LIN {E6POS: X 1201.000, Y -192.200, Z 553.000, A 0.000, B 90.000, C 0.000, E1 0.000, E2 0.0, E3 0.0, E4 0.0, E5 0.0, E6 0.0} C_DIS
LIN {E6POS: X 1201.000, Y -191.200, Z 553.000, A 0.000, B 90.000, C 0.000, E1 0.000, E2 0.0, E3 0.0, E4 0.0, E5 0.0, E6 0.0} C_DIS
LIN {E6POS: X 1201.000, Y -190.200, Z 553.000, A 0.000, B 90.000, C 0.000, E1 0.000, E2 0.0, E3 0.0, E4 0.0, E5 0.0, E6 0.0} C_DIS
LIN {E6POS: X 1201.000, Y -189.200, Z 553.000, A 0.000, B 90.000, C 0.000, E1 0.000, E2 0.0, E3 0.0, E4 0.0, E5 0.0, E6 0.0} C_DIS
LIN {E6POS: X 1201.000, Y -188.200, Z 553.000, A 0.000, B 90.000, C 0.000, E1 0.000, E2 0.0, E3 0.0, E4 0.0, E5 0.0, E6 0.0} C_DIS
LIN {E6POS: X 1201.000, Y -187.200, Z 553.000, A 0.000, B 90.000, C 0.000, E1 0.000, E2 0.0, E3 0.0, E4 0.0, E5 0.0, E6 0.0} C_DIS
LIN {E6POS: X 1201.000, Y -187.200, Z 553.000, A 0.000, B 90.000, C 0.000, E1 0.000, E2 0.0, E3 0.0, E4 0.0, E5 0.0, E6 0.0} C_DIS
LIN {E6POS: X 1200.000, Y -187.200, Z 553.000, A 0.000, B 90.000, C 0.000, E1 0.000, E2 0.0, E3 0.0, E4 0.0, E5 0.0, E6 0.0} C_DIS
LIN {E6POS: X 1199.000, Y -187.200, Z 553.000, A 0.000, B 90.000, C 0.000, E1 0.000, E2 0.0, E3 0.0, E4 0.0, E5 0.0, E6 0.0} C_DIS
LIN {E6POS: X 1198.000, Y -187.200, Z 553.000, A 0.000, B 90.000, C 0.000, E1 0.000, E2 0.0, E3 0.0, E4 0.0, E5 0.0, E6 0.0} C_DIS
LIN {E6POS: X 1197.000, Y -187.200, Z 553.000, A 0.000, B 90.000, C 0.000, E1 0.000, E2 0.0, E3 0.0, E4 0.0, E5 0.0, E6 0.0} C_DIS
LIN {E6POS: X 1196.000, Y -187.200, Z 553.000, A 0.000, B 90.000, C 0.000, E1 0.000, E2 0.0, E3 0.0, E4 0.0, E5 0.0, E6 0.0} C_DIS
LIN {E6POS: X 1196.000, Y -187.200, Z 553.000, A 0.000, B 90.000, C 0.000, E1 0.000, E2 0.0, E3 0.0, E4 0.0, E5 0.0, E6 0.0} C_DIS
LIN {E6POS: X 1196.000, Y -188.200, Z 553.000, A 0.000, B 90.000, C 0.000, E1 0.000, E2 0.0, E3 0.0, E4 0.0, E5 0.0, E6 0.0} C_DIS
LIN {E6POS: X 1196.000, Y -189.200, Z 553.000, A 0.000, B 90.000, C 0.000, E1 0.000, E2 0.0, E3 0.0, E4 0.0, E5 0.0, E6 0.0} C_DIS
LIN {E6POS: X 1196.000, Y -190.200, Z 553.000, A 0.000, B 90.000, C 0.000, E1 0.000, E2 0.0, E3 0.0, E4 0.0, E5 0.0, E6 0.0} C_DIS
LIN {E6POS: X 1196.000, Y -191.200, Z 553.000, A 0.000, B 90.000, C 0.000, E1 0.000, E2 0.0, E3 0.0, E4 0.0, E5 0.0, E6 0.0} C_DIS
LIN {E6POS: X 1196.000, Y -192.200, Z 553.000, A 0.000, B 90.000, C 0.000, E1 0.000, E2 0.0, E3 0.0, E4 0.0, E5 0.0, E6 0.0} C_DIS
LIN {E6POS: X 1196.000, Y -193.200, Z 553.000, A 0.000, B 90.000, C 0.000, E1 0.000, E2 0.0, E3 0.0, E4 0.0, E5 0.0, E6 0.0} C_DIS
LIN {E6POS: X 1196.000, Y -194.200, Z 553.000, A 0.000, B 90.000, C 0.000, E1 0.000, E2 0.0, E3 0.0, E4 0.0, E5 0.0, E6 0.0} C_DIS
LIN {E6POS: X 1196.000, Y -195.200, Z 553.000, A 0.000, B 90.000, C 0.000, E1 0.000, E2 0.0, E3 0.0, E4 0.0, E5 0.0, E6 0.0} C_DIS
LIN {E6POS: X 1196.000, Y -196.200, Z 553.000, A 0.000, B 90.000, C 0.000, E1 0.000, E2 0.0, E3 0.0, E4 0.0, E5 0.0, E6 0.0} C_DIS
LIN {E6POS: X 1196.000, Y -197.200, Z 553.000, A 0.000, B 90.000, C 0.000, E1 0.000, E2 0.0, E3 0.0, E4 0.0, E5 0.0, E6 0.0} C_DIS
LIN {E6POS: X 1196.000, Y -198.200, Z 553.000, A 0.000, B 90.000, C 0.000, E1 0.000, E2 0.0, E3 0.0, E4 0.0, E5 0.0, E6 0.0} C_DIS
LIN {E6POS: X 1196.000, Y -199.200, Z 553.000, A 0.000, B 90.000, C 0.000, E1 0.000, E2 0.0, E3 0.0, E4 0.0, E5 0.0, E6 0.0} C_DIS
LIN {E6POS: X 1196.000, Y -200.200, Z 553.000, A 0.000, B 90.000, C 0.000, E1 0.000, E2 0.0, E3 0.0, E4 0.0, E5 0.0, E6 0.0} C_DIS
LIN {E6POS: X 1196.000, Y -201.200, Z 553.000, A 0.000, B 90.000, C 0.000, E1 0.000, E2 0.0, E3 0.0, E4 0.0, E5 0.0, E6 0.0} C_DIS
LIN {E6POS: X 1196.000, Y -202.200, Z 553.000, A 0.000, B 90.000, C 0.000, E1 0.000, E2 0.0, E3 0.0, E4 0.0, E5 0.0, E6 0.0} C_DIS
LIN {E6POS: X 1196.000, Y -203.200, Z 553.000, A 0.000, B 90.000, C 0.000, E1 0.000, E2 0.0, E3 0.0, E4 0.0, E5 0.0, E6 0.0} C_DIS
LIN {E6POS: X 1196.000, Y -204.200, Z 553.000, A 0.000, B 90.000, C 0.000, E1 0.000, E2 0.0, E3 0.0, E4 0.0, E5 0.0, E6 0.0} C_DIS
LIN {E6POS: X 1196.000, Y -205.200, Z 553.000, A 0.000, B 90.000, C 0.000, E1 0.000, E2 0.0, E3 0.0, E4 0.0, E5 0.0, E6 0.0} C_DIS
LIN {E6POS: X 1196.000, Y -206.200, Z 553.000, A 0.000, B 90.000, C 0.000, E1 0.000, E2 0.0, E3 0.0, E4 0.0, E5 0.0, E6 0.0} C_DIS
LIN {E6POS: X 1196.000, Y -207.200, Z 553.000, A 0.000, B 90.000, C 0.000, E1 0.000, E2 0.0, E3 0.0, E4 0.0, E5 0.0, E6 0.0} C_DIS
LIN {E6POS: X 1196.000, Y -208.200, Z 553.000, A 0.000, B 90.000, C 0.000, E1 0.000, E2 0.0, E3 0.0, E4 0.0, E5 0.0, E6 0.0} C_DIS
LIN {E6POS: X 1196.000, Y -209.200, Z 553.000, A 0.000, B 90.000, C 0.000, E1 0.000, E2 0.0, E3 0.0, E4 0.0, E5 0.0, E6 0.0} C_DIS
LIN {E6POS: X 1196.000, Y -210.200, Z 553.000, A 0.000, B 90.000, C 0.000, E1 0.000, E2 0.0, E3 0.0, E4 0.0, E5 0.0, E6 0.0} C_DIS
LIN {E6POS: X 1196.000, Y -211.200, Z 553.000, A 0.000, B 90.000, C 0.000, E1 0.000, E2 0.0, E3 0.0, E4 0.0, E5 0.0, E6 0.0} C_DIS
LIN {E6POS: X 1196.000, Y -212.200, Z 553.000, A 0.000, B 90.000, C 0.000, E1 0.000, E2 0.0, E3 0.0, E4 0.0, E5 0.0, E6 0.0} C_DIS
LIN {E6POS: X 1196.000, Y -213.200, Z 553.000, A 0.000, B 90.000, C 0.000, E1 0.000, E2 0.0, E3 0.0, E4 0.0, E5 0.0, E6 0.0} C_DIS
LIN {E6POS: X 1196.000, Y -214.200, Z 553.000, A 0.000, B 90.000, C 0.000, E1 0.000, E2 0.0, E3 0.0, E4 0.0, E5 0.0, E6 0.0} C_DIS
LIN {E6POS: X 1196.000, Y -215.200, Z 553.000, A 0.000, B 90.000, C 0.000, E1 0.000, E2 0.0, E3 0.0, E4 0.0, E5 0.0, E6 0.0} C_DIS
LIN {E6POS: X 1196.000, Y -216.200, Z 553.000, A 0.000, B 90.000, C 0.000, E1 0.000, E2 0.0, E3 0.0, E4 0.0, E5 0.0, E6 0.0} C_DIS
LIN {E6POS: X 1196.000, Y -217.200, Z 553.000, A 0.000, B 90.000, C 0.000, E1 0.000, E2 0.0, E3 0.0, E4 0.0, E5 0.0, E6 0.0} C_DIS
LIN {E6POS: X 1196.000, Y -218.200, Z 553.000, A 0.000, B 90.000, C 0.000, E1 0.000, E2 0.0, E3 0.0, E4 0.0, E5 0.0, E6 0.0} C_DIS
LIN {E6POS: X 1196.000, Y -219.200, Z 553.000, A 0.000, B 90.000, C 0.000, E1 0.000, E2 0.0, E3 0.0, E4 0.0, E5 0.0, E6 0.0} C_DIS
LIN {E6POS: X 1196.000, Y -220.200, Z 553.000, A 0.000, B 90.000, C 0.000, E1 0.000, E2 0.0, E3 0.0, E4 0.0, E5 0.0, E6 0.0} C_DIS
LIN {E6POS: X 1196.000, Y -221.200, Z 553.000, A 0.000, B 90.000, C 0.000, E1 0.000, E2 0.0, E3 0.0, E4 0.0, E5 0.0, E6 0.0} C_DIS
LIN {E6POS: X 1196.000, Y -222.200, Z 553.000, A 0.000, B 90.000, C 0.000, E1 0.000, E2 0.0, E3 0.0, E4 0.0, E5 0.0, E6 0.0} C_DIS
LIN {E6POS: X 1196.000, Y -223.200, Z 553.000, A 0.000, B 90.000, C 0.000, E1 0.000, E2 0.0, E3 0.0, E4 0.0, E5 0.0, E6 0.0} C_DIS
LIN {E6POS: X 1196.000, Y -224.200, Z 553.000, A 0.000, B 90.000, C 0.000, E1 0.000, E2 0.0, E3 0.0, E4 0.0, E5 0.0, E6 0.0} C_DIS
LIN {E6POS: X 1196.000, Y -225.200, Z 553.000, A 0.000, B 90.000, C 0.000, E1 0.000, E2 0.0, E3 0.0, E4 0.0, E5 0.0, E6 0.0} C_DIS
LIN {E6POS: X 1196.000, Y -226.200, Z 553.000, A 0.000, B 90.000, C 0.000, E1 0.000, E2 0.0, E3 0.0, E4 0.0, E5 0.0, E6 0.0} C_DIS
LIN {E6POS: X 1196.000, Y -227.200, Z 553.000, A 0.000, B 90.000, C 0.000, E1 0.000, E2 0.0, E3 0.0, E4 0.0, E5 0.0, E6 0.0} C_DIS
LIN {E6POS: X 1196.000, Y -228.200, Z 553.000, A 0.000, B 90.000, C 0.000, E1 0.000, E2 0.0, E3 0.0, E4 0.0, E5 0.0, E6 0.0} C_DIS
LIN {E6POS: X 1196.000, Y -229.200, Z 553.000, A 0.000, B 90.000, C 0.000, E1 0.000, E2 0.0, E3 0.0, E4 0.0, E5 0.0, E6 0.0} C_DIS
LIN {E6POS: X 1196.000, Y -230.200, Z 553.000, A 0.000, B 90.000, C 0.000, E1 0.000, E2 0.0, E3 0.0, E4 0.0, E5 0.0, E6 0.0} C_DIS
LIN {E6POS: X 1196.000, Y -231.200, Z 553.000, A 0.000, B 90.000, C 0.000, E1 0.000, E2 0.0, E3 0.0, E4 0.0, E5 0.0, E6 0.0} C_DIS
LIN {E6POS: X 1196.000, Y -232.200, Z 553.000, A 0.000, B 90.000, C 0.000, E1 0.000, E2 0.0, E3 0.0, E4 0.0, E5 0.0, E6 0.0} C_DIS
LIN {E6POS: X 1196.000, Y -233.200, Z 553.000, A 0.000, B 90.000, C 0.000, E1 0.000, E2 0.0, E3 0.0, E4 0.0, E5 0.0, E6 0.0} C_DIS
LIN {E6POS: X 1196.000, Y -234.200, Z 553.000, A 0.000, B 90.000, C 0.000, E1 0.000, E2 0.0, E3 0.0, E4 0.0, E5 0.0, E6 0.0} C_DIS
LIN {E6POS: X 1196.000, Y -235.200, Z 553.000, A 0.000, B 90.000, C 0.000, E1 0.000, E2 0.0, E3 0.0, E4 0.0, E5 0.0, E6 0.0} C_DIS
LIN {E6POS: X 1196.000, Y -236.200, Z 553.000, A 0.000, B 90.000, C 0.000, E1 0.000, E2 0.0, E3 0.0, E4 0.0, E5 0.0, E6 0.0} C_DIS
LIN {E6POS: X 1196.000, Y -237.200, Z 553.000, A 0.000, B 90.000, C 0.000, E1 0.000, E2 0.0, E3 0.0, E4 0.0, E5 0.0, E6 0.0} C_DIS
LIN {E6POS: X 1196.000, Y -237.200, Z 554.000, A 0.000, B 90.000, C 0.000, E1 0.000, E2 0.0, E3 0.0, E4 0.0, E5 0.0, E6 0.0} C_DIS
LIN {E6POS: X 1197.000, Y -237.200, Z 554.000, A 0.000, B 90.000, C 0.000, E1 0.000, E2 0.0, E3 0.0, E4 0.0, E5 0.0, E6 0.0} C_DIS
LIN {E6POS: X 1198.000, Y -237.200, Z 554.000, A 0.000, B 90.000, C 0.000, E1 0.000, E2 0.0, E3 0.0, E4 0.0, E5 0.0, E6 0.0} C_DIS
LIN {E6POS: X 1199.000, Y -237.200, Z 554.000, A 0.000, B 90.000, C 0.000, E1 0.000, E2 0.0, E3 0.0, E4 0.0, E5 0.0, E6 0.0} C_DIS
LIN {E6POS: X 1200.000, Y -237.200, Z 554.000, A 0.000, B 90.000, C 0.000, E1 0.000, E2 0.0, E3 0.0, E4 0.0, E5 0.0, E6 0.0} C_DIS
LIN {E6POS: X 1201.000, Y -237.200, Z 554.000, A 0.000, B 90.000, C 0.000, E1 0.000, E2 0.0, E3 0.0, E4 0.0, E5 0.0, E6 0.0} C_DIS
LIN {E6POS: X 1201.000, Y -237.200, Z 554.000, A 0.000, B 90.000, C 0.000, E1 0.000, E2 0.0, E3 0.0, E4 0.0, E5 0.0, E6 0.0} C_DIS
LIN {E6POS: X 1201.000, Y -236.200, Z 554.000, A 0.000, B 90.000, C 0.000, E1 0.000, E2 0.0, E3 0.0, E4 0.0, E5 0.0, E6 0.0} C_DIS
LIN {E6POS: X 1201.000, Y -235.200, Z 554.000, A 0.000, B 90.000, C 0.000, E1 0.000, E2 0.0, E3 0.0, E4 0.0, E5 0.0, E6 0.0} C_DIS
LIN {E6POS: X 1201.000, Y -234.200, Z 554.000, A 0.000, B 90.000, C 0.000, E1 0.000, E2 0.0, E3 0.0, E4 0.0, E5 0.0, E6 0.0} C_DIS
LIN {E6POS: X 1201.000, Y -233.200, Z 554.000, A 0.000, B 90.000, C 0.000, E1 0.000, E2 0.0, E3 0.0, E4 0.0, E5 0.0, E6 0.0} C_DIS
LIN {E6POS: X 1201.000, Y -232.200, Z 554.000, A 0.000, B 90.000, C 0.000, E1 0.000, E2 0.0, E3 0.0, E4 0.0, E5 0.0, E6 0.0} C_DIS
LIN {E6POS: X 1201.000, Y -231.200, Z 554.000, A 0.000, B 90.000, C 0.000, E1 0.000, E2 0.0, E3 0.0, E4 0.0, E5 0.0, E6 0.0} C_DIS
LIN {E6POS: X 1201.000, Y -230.200, Z 554.000, A 0.000, B 90.000, C 0.000, E1 0.000, E2 0.0, E3 0.0, E4 0.0, E5 0.0, E6 0.0} C_DIS
LIN {E6POS: X 1201.000, Y -229.200, Z 554.000, A 0.000, B 90.000, C 0.000, E1 0.000, E2 0.0, E3 0.0, E4 0.0, E5 0.0, E6 0.0} C_DIS
LIN {E6POS: X 1201.000, Y -228.200, Z 554.000, A 0.000, B 90.000, C 0.000, E1 0.000, E2 0.0, E3 0.0, E4 0.0, E5 0.0, E6 0.0} C_DIS
LIN {E6POS: X 1201.000, Y -227.200, Z 554.000, A 0.000, B 90.000, C 0.000, E1 0.000, E2 0.0, E3 0.0, E4 0.0, E5 0.0, E6 0.0} C_DIS
LIN {E6POS: X 1201.000, Y -226.200, Z 554.000, A 0.000, B 90.000, C 0.000, E1 0.000, E2 0.0, E3 0.0, E4 0.0, E5 0.0, E6 0.0} C_DIS
LIN {E6POS: X 1201.000, Y -225.200, Z 554.000, A 0.000, B 90.000, C 0.000, E1 0.000, E2 0.0, E3 0.0, E4 0.0, E5 0.0, E6 0.0} C_DIS
LIN {E6POS: X 1201.000, Y -224.200, Z 554.000, A 0.000, B 90.000, C 0.000, E1 0.000, E2 0.0, E3 0.0, E4 0.0, E5 0.0, E6 0.0} C_DIS
LIN {E6POS: X 1201.000, Y -223.200, Z 554.000, A 0.000, B 90.000, C 0.000, E1 0.000, E2 0.0, E3 0.0, E4 0.0, E5 0.0, E6 0.0} C_DIS
LIN {E6POS: X 1201.000, Y -222.200, Z 554.000, A 0.000, B 90.000, C 0.000, E1 0.000, E2 0.0, E3 0.0, E4 0.0, E5 0.0, E6 0.0} C_DIS
LIN {E6POS: X 1201.000, Y -221.200, Z 554.000, A 0.000, B 90.000, C 0.000, E1 0.000, E2 0.0, E3 0.0, E4 0.0, E5 0.0, E6 0.0} C_DIS
LIN {E6POS: X 1201.000, Y -220.200, Z 554.000, A 0.000, B 90.000, C 0.000, E1 0.000, E2 0.0, E3 0.0, E4 0.0, E5 0.0, E6 0.0} C_DIS
LIN {E6POS: X 1201.000, Y -219.200, Z 554.000, A 0.000, B 90.000, C 0.000, E1 0.000, E2 0.0, E3 0.0, E4 0.0, E5 0.0, E6 0.0} C_DIS
LIN {E6POS: X 1201.000, Y -218.200, Z 554.000, A 0.000, B 90.000, C 0.000, E1 0.000, E2 0.0, E3 0.0, E4 0.0, E5 0.0, E6 0.0} C_DIS
LIN {E6POS: X 1201.000, Y -217.200, Z 554.000, A 0.000, B 90.000, C 0.000, E1 0.000, E2 0.0, E3 0.0, E4 0.0, E5 0.0, E6 0.0} C_DIS
LIN {E6POS: X 1201.000, Y -216.200, Z 554.000, A 0.000, B 90.000, C 0.000, E1 0.000, E2 0.0, E3 0.0, E4 0.0, E5 0.0, E6 0.0} C_DIS
LIN {E6POS: X 1201.000, Y -215.200, Z 554.000, A 0.000, B 90.000, C 0.000, E1 0.000, E2 0.0, E3 0.0, E4 0.0, E5 0.0, E6 0.0} C_DIS
LIN {E6POS: X 1201.000, Y -214.200, Z 554.000, A 0.000, B 90.000, C 0.000, E1 0.000, E2 0.0, E3 0.0, E4 0.0, E5 0.0, E6 0.0} C_DIS
LIN {E6POS: X 1201.000, Y -213.200, Z 554.000, A 0.000, B 90.000, C 0.000, E1 0.000, E2 0.0, E3 0.0, E4 0.0, E5 0.0, E6 0.0} C_DIS
LIN {E6POS: X 1201.000, Y -212.200, Z 554.000, A 0.000, B 90.000, C 0.000, E1 0.000, E2 0.0, E3 0.0, E4 0.0, E5 0.0, E6 0.0} C_DIS
LIN {E6POS: X 1201.000, Y -211.200, Z 554.000, A 0.000, B 90.000, C 0.000, E1 0.000, E2 0.0, E3 0.0, E4 0.0, E5 0.0, E6 0.0} C_DIS
LIN {E6POS: X 1201.000, Y -210.200, Z 554.000, A 0.000, B 90.000, C 0.000, E1 0.000, E2 0.0, E3 0.0, E4 0.0, E5 0.0, E6 0.0} C_DIS
LIN {E6POS: X 1201.000, Y -209.200, Z 554.000, A 0.000, B 90.000, C 0.000, E1 0.000, E2 0.0, E3 0.0, E4 0.0, E5 0.0, E6 0.0} C_DIS
LIN {E6POS: X 1201.000, Y -208.200, Z 554.000, A 0.000, B 90.000, C 0.000, E1 0.000, E2 0.0, E3 0.0, E4 0.0, E5 0.0, E6 0.0} C_DIS
LIN {E6POS: X 1201.000, Y -207.200, Z 554.000, A 0.000, B 90.000, C 0.000, E1 0.000, E2 0.0, E3 0.0, E4 0.0, E5 0.0, E6 0.0} C_DIS
LIN {E6POS: X 1201.000, Y -206.200, Z 554.000, A 0.000, B 90.000, C 0.000, E1 0.000, E2 0.0, E3 0.0, E4 0.0, E5 0.0, E6 0.0} C_DIS
LIN {E6POS: X 1201.000, Y -205.200, Z 554.000, A 0.000, B 90.000, C 0.000, E1 0.000, E2 0.0, E3 0.0, E4 0.0, E5 0.0, E6 0.0} C_DIS
LIN {E6POS: X 1201.000, Y -204.200, Z 554.000, A 0.000, B 90.000, C 0.000, E1 0.000, E2 0.0, E3 0.0, E4 0.0, E5 0.0, E6 0.0} C_DIS
LIN {E6POS: X 1201.000, Y -203.200, Z 554.000, A 0.000, B 90.000, C 0.000, E1 0.000, E2 0.0, E3 0.0, E4 0.0, E5 0.0, E6 0.0} C_DIS
LIN {E6POS: X 1201.000, Y -202.200, Z 554.000, A 0.000, B 90.000, C 0.000, E1 0.000, E2 0.0, E3 0.0, E4 0.0, E5 0.0, E6 0.0} C_DIS
LIN {E6POS: X 1201.000, Y -201.200, Z 554.000, A 0.000, B 90.000, C 0.000, E1 0.000, E2 0.0, E3 0.0, E4 0.0, E5 0.0, E6 0.0} C_DIS
LIN {E6POS: X 1201.000, Y -200.200, Z 554.000, A 0.000, B 90.000, C 0.000, E1 0.000, E2 0.0, E3 0.0, E4 0.0, E5 0.0, E6 0.0} C_DIS
LIN {E6POS: X 1201.000, Y -199.200, Z 554.000, A 0.000, B 90.000, C 0.000, E1 0.000, E2 0.0, E3 0.0, E4 0.0, E5 0.0, E6 0.0} C_DIS
LIN {E6POS: X 1201.000, Y -198.200, Z 554.000, A 0.000, B 90.000, C 0.000, E1 0.000, E2 0.0, E3 0.0, E4 0.0, E5 0.0, E6 0.0} C_DIS
LIN {E6POS: X 1201.000, Y -197.200, Z 554.000, A 0.000, B 90.000, C 0.000, E1 0.000, E2 0.0, E3 0.0, E4 0.0, E5 0.0, E6 0.0} C_DIS
LIN {E6POS: X 1201.000, Y -196.200, Z 554.000, A 0.000, B 90.000, C 0.000, E1 0.000, E2 0.0, E3 0.0, E4 0.0, E5 0.0, E6 0.0} C_DIS
LIN {E6POS: X 1201.000, Y -195.200, Z 554.000, A 0.000, B 90.000, C 0.000, E1 0.000, E2 0.0, E3 0.0, E4 0.0, E5 0.0, E6 0.0} C_DIS
LIN {E6POS: X 1201.000, Y -194.200, Z 554.000, A 0.000, B 90.000, C 0.000, E1 0.000, E2 0.0, E3 0.0, E4 0.0, E5 0.0, E6 0.0} C_DIS
LIN {E6POS: X 1201.000, Y -193.200, Z 554.000, A 0.000, B 90.000, C 0.000, E1 0.000, E2 0.0, E3 0.0, E4 0.0, E5 0.0, E6 0.0} C_DIS
LIN {E6POS: X 1201.000, Y -192.200, Z 554.000, A 0.000, B 90.000, C 0.000, E1 0.000, E2 0.0, E3 0.0, E4 0.0, E5 0.0, E6 0.0} C_DIS
LIN {E6POS: X 1201.000, Y -191.200, Z 554.000, A 0.000, B 90.000, C 0.000, E1 0.000, E2 0.0, E3 0.0, E4 0.0, E5 0.0, E6 0.0} C_DIS
LIN {E6POS: X 1201.000, Y -190.200, Z 554.000, A 0.000, B 90.000, C 0.000, E1 0.000, E2 0.0, E3 0.0, E4 0.0, E5 0.0, E6 0.0} C_DIS
LIN {E6POS: X 1201.000, Y -189.200, Z 554.000, A 0.000, B 90.000, C 0.000, E1 0.000, E2 0.0, E3 0.0, E4 0.0, E5 0.0, E6 0.0} C_DIS
LIN {E6POS: X 1201.000, Y -188.200, Z 554.000, A 0.000, B 90.000, C 0.000, E1 0.000, E2 0.0, E3 0.0, E4 0.0, E5 0.0, E6 0.0} C_DIS
LIN {E6POS: X 1201.000, Y -187.200, Z 554.000, A 0.000, B 90.000, C 0.000, E1 0.000, E2 0.0, E3 0.0, E4 0.0, E5 0.0, E6 0.0} C_DIS
LIN {E6POS: X 1201.000, Y -187.200, Z 554.000, A 0.000, B 90.000, C 0.000, E1 0.000, E2 0.0, E3 0.0, E4 0.0, E5 0.0, E6 0.0} C_DIS
LIN {E6POS: X 1200.000, Y -187.200, Z 554.000, A 0.000, B 90.000, C 0.000, E1 0.000, E2 0.0, E3 0.0, E4 0.0, E5 0.0, E6 0.0} C_DIS
LIN {E6POS: X 1199.000, Y -187.200, Z 554.000, A 0.000, B 90.000, C 0.000, E1 0.000, E2 0.0, E3 0.0, E4 0.0, E5 0.0, E6 0.0} C_DIS
LIN {E6POS: X 1198.000, Y -187.200, Z 554.000, A 0.000, B 90.000, C 0.000, E1 0.000, E2 0.0, E3 0.0, E4 0.0, E5 0.0, E6 0.0} C_DIS
LIN {E6POS: X 1197.000, Y -187.200, Z 554.000, A 0.000, B 90.000, C 0.000, E1 0.000, E2 0.0, E3 0.0, E4 0.0, E5 0.0, E6 0.0} C_DIS
LIN {E6POS: X 1196.000, Y -187.200, Z 554.000, A 0.000, B 90.000, C 0.000, E1 0.000, E2 0.0, E3 0.0, E4 0.0, E5 0.0, E6 0.0} C_DIS
LIN {E6POS: X 1196.000, Y -187.200, Z 554.000, A 0.000, B 90.000, C 0.000, E1 0.000, E2 0.0, E3 0.0, E4 0.0, E5 0.0, E6 0.0} C_DIS
LIN {E6POS: X 1196.000, Y -188.200, Z 554.000, A 0.000, B 90.000, C 0.000, E1 0.000, E2 0.0, E3 0.0, E4 0.0, E5 0.0, E6 0.0} C_DIS
LIN {E6POS: X 1196.000, Y -189.200, Z 554.000, A 0.000, B 90.000, C 0.000, E1 0.000, E2 0.0, E3 0.0, E4 0.0, E5 0.0, E6 0.0} C_DIS
LIN {E6POS: X 1196.000, Y -190.200, Z 554.000, A 0.000, B 90.000, C 0.000, E1 0.000, E2 0.0, E3 0.0, E4 0.0, E5 0.0, E6 0.0} C_DIS
LIN {E6POS: X 1196.000, Y -191.200, Z 554.000, A 0.000, B 90.000, C 0.000, E1 0.000, E2 0.0, E3 0.0, E4 0.0, E5 0.0, E6 0.0} C_DIS
LIN {E6POS: X 1196.000, Y -192.200, Z 554.000, A 0.000, B 90.000, C 0.000, E1 0.000, E2 0.0, E3 0.0, E4 0.0, E5 0.0, E6 0.0} C_DIS
LIN {E6POS: X 1196.000, Y -193.200, Z 554.000, A 0.000, B 90.000, C 0.000, E1 0.000, E2 0.0, E3 0.0, E4 0.0, E5 0.0, E6 0.0} C_DIS
LIN {E6POS: X 1196.000, Y -194.200, Z 554.000, A 0.000, B 90.000, C 0.000, E1 0.000, E2 0.0, E3 0.0, E4 0.0, E5 0.0, E6 0.0} C_DIS
LIN {E6POS: X 1196.000, Y -195.200, Z 554.000, A 0.000, B 90.000, C 0.000, E1 0.000, E2 0.0, E3 0.0, E4 0.0, E5 0.0, E6 0.0} C_DIS
LIN {E6POS: X 1196.000, Y -196.200, Z 554.000, A 0.000, B 90.000, C 0.000, E1 0.000, E2 0.0, E3 0.0, E4 0.0, E5 0.0, E6 0.0} C_DIS
LIN {E6POS: X 1196.000, Y -197.200, Z 554.000, A 0.000, B 90.000, C 0.000, E1 0.000, E2 0.0, E3 0.0, E4 0.0, E5 0.0, E6 0.0} C_DIS
LIN {E6POS: X 1196.000, Y -198.200, Z 554.000, A 0.000, B 90.000, C 0.000, E1 0.000, E2 0.0, E3 0.0, E4 0.0, E5 0.0, E6 0.0} C_DIS
LIN {E6POS: X 1196.000, Y -199.200, Z 554.000, A 0.000, B 90.000, C 0.000, E1 0.000, E2 0.0, E3 0.0, E4 0.0, E5 0.0, E6 0.0} C_DIS
LIN {E6POS: X 1196.000, Y -200.200, Z 554.000, A 0.000, B 90.000, C 0.000, E1 0.000, E2 0.0, E3 0.0, E4 0.0, E5 0.0, E6 0.0} C_DIS
LIN {E6POS: X 1196.000, Y -201.200, Z 554.000, A 0.000, B 90.000, C 0.000, E1 0.000, E2 0.0, E3 0.0, E4 0.0, E5 0.0, E6 0.0} C_DIS
LIN {E6POS: X 1196.000, Y -202.200, Z 554.000, A 0.000, B 90.000, C 0.000, E1 0.000, E2 0.0, E3 0.0, E4 0.0, E5 0.0, E6 0.0} C_DIS
LIN {E6POS: X 1196.000, Y -203.200, Z 554.000, A 0.000, B 90.000, C 0.000, E1 0.000, E2 0.0, E3 0.0, E4 0.0, E5 0.0, E6 0.0} C_DIS
LIN {E6POS: X 1196.000, Y -204.200, Z 554.000, A 0.000, B 90.000, C 0.000, E1 0.000, E2 0.0, E3 0.0, E4 0.0, E5 0.0, E6 0.0} C_DIS
LIN {E6POS: X 1196.000, Y -205.200, Z 554.000, A 0.000, B 90.000, C 0.000, E1 0.000, E2 0.0, E3 0.0, E4 0.0, E5 0.0, E6 0.0} C_DIS
LIN {E6POS: X 1196.000, Y -206.200, Z 554.000, A 0.000, B 90.000, C 0.000, E1 0.000, E2 0.0, E3 0.0, E4 0.0, E5 0.0, E6 0.0} C_DIS
LIN {E6POS: X 1196.000, Y -207.200, Z 554.000, A 0.000, B 90.000, C 0.000, E1 0.000, E2 0.0, E3 0.0, E4 0.0, E5 0.0, E6 0.0} C_DIS
LIN {E6POS: X 1196.000, Y -208.200, Z 554.000, A 0.000, B 90.000, C 0.000, E1 0.000, E2 0.0, E3 0.0, E4 0.0, E5 0.0, E6 0.0} C_DIS
LIN {E6POS: X 1196.000, Y -209.200, Z 554.000, A 0.000, B 90.000, C 0.000, E1 0.000, E2 0.0, E3 0.0, E4 0.0, E5 0.0, E6 0.0} C_DIS
LIN {E6POS: X 1196.000, Y -210.200, Z 554.000, A 0.000, B 90.000, C 0.000, E1 0.000, E2 0.0, E3 0.0, E4 0.0, E5 0.0, E6 0.0} C_DIS
LIN {E6POS: X 1196.000, Y -211.200, Z 554.000, A 0.000, B 90.000, C 0.000, E1 0.000, E2 0.0, E3 0.0, E4 0.0, E5 0.0, E6 0.0} C_DIS
LIN {E6POS: X 1196.000, Y -212.200, Z 554.000, A 0.000, B 90.000, C 0.000, E1 0.000, E2 0.0, E3 0.0, E4 0.0, E5 0.0, E6 0.0} C_DIS
LIN {E6POS: X 1196.000, Y -213.200, Z 554.000, A 0.000, B 90.000, C 0.000, E1 0.000, E2 0.0, E3 0.0, E4 0.0, E5 0.0, E6 0.0} C_DIS
LIN {E6POS: X 1196.000, Y -214.200, Z 554.000, A 0.000, B 90.000, C 0.000, E1 0.000, E2 0.0, E3 0.0, E4 0.0, E5 0.0, E6 0.0} C_DIS
LIN {E6POS: X 1196.000, Y -215.200, Z 554.000, A 0.000, B 90.000, C 0.000, E1 0.000, E2 0.0, E3 0.0, E4 0.0, E5 0.0, E6 0.0} C_DIS
LIN {E6POS: X 1196.000, Y -216.200, Z 554.000, A 0.000, B 90.000, C 0.000, E1 0.000, E2 0.0, E3 0.0, E4 0.0, E5 0.0, E6 0.0} C_DIS
LIN {E6POS: X 1196.000, Y -217.200, Z 554.000, A 0.000, B 90.000, C 0.000, E1 0.000, E2 0.0, E3 0.0, E4 0.0, E5 0.0, E6 0.0} C_DIS
LIN {E6POS: X 1196.000, Y -218.200, Z 554.000, A 0.000, B 90.000, C 0.000, E1 0.000, E2 0.0, E3 0.0, E4 0.0, E5 0.0, E6 0.0} C_DIS
LIN {E6POS: X 1196.000, Y -219.200, Z 554.000, A 0.000, B 90.000, C 0.000, E1 0.000, E2 0.0, E3 0.0, E4 0.0, E5 0.0, E6 0.0} C_DIS
LIN {E6POS: X 1196.000, Y -220.200, Z 554.000, A 0.000, B 90.000, C 0.000, E1 0.000, E2 0.0, E3 0.0, E4 0.0, E5 0.0, E6 0.0} C_DIS
LIN {E6POS: X 1196.000, Y -221.200, Z 554.000, A 0.000, B 90.000, C 0.000, E1 0.000, E2 0.0, E3 0.0, E4 0.0, E5 0.0, E6 0.0} C_DIS
LIN {E6POS: X 1196.000, Y -222.200, Z 554.000, A 0.000, B 90.000, C 0.000, E1 0.000, E2 0.0, E3 0.0, E4 0.0, E5 0.0, E6 0.0} C_DIS
LIN {E6POS: X 1196.000, Y -223.200, Z 554.000, A 0.000, B 90.000, C 0.000, E1 0.000, E2 0.0, E3 0.0, E4 0.0, E5 0.0, E6 0.0} C_DIS
LIN {E6POS: X 1196.000, Y -224.200, Z 554.000, A 0.000, B 90.000, C 0.000, E1 0.000, E2 0.0, E3 0.0, E4 0.0, E5 0.0, E6 0.0} C_DIS
LIN {E6POS: X 1196.000, Y -225.200, Z 554.000, A 0.000, B 90.000, C 0.000, E1 0.000, E2 0.0, E3 0.0, E4 0.0, E5 0.0, E6 0.0} C_DIS
LIN {E6POS: X 1196.000, Y -226.200, Z 554.000, A 0.000, B 90.000, C 0.000, E1 0.000, E2 0.0, E3 0.0, E4 0.0, E5 0.0, E6 0.0} C_DIS
LIN {E6POS: X 1196.000, Y -227.200, Z 554.000, A 0.000, B 90.000, C 0.000, E1 0.000, E2 0.0, E3 0.0, E4 0.0, E5 0.0, E6 0.0} C_DIS
LIN {E6POS: X 1196.000, Y -228.200, Z 554.000, A 0.000, B 90.000, C 0.000, E1 0.000, E2 0.0, E3 0.0, E4 0.0, E5 0.0, E6 0.0} C_DIS
LIN {E6POS: X 1196.000, Y -229.200, Z 554.000, A 0.000, B 90.000, C 0.000, E1 0.000, E2 0.0, E3 0.0, E4 0.0, E5 0.0, E6 0.0} C_DIS
LIN {E6POS: X 1196.000, Y -230.200, Z 554.000, A 0.000, B 90.000, C 0.000, E1 0.000, E2 0.0, E3 0.0, E4 0.0, E5 0.0, E6 0.0} C_DIS
LIN {E6POS: X 1196.000, Y -231.200, Z 554.000, A 0.000, B 90.000, C 0.000, E1 0.000, E2 0.0, E3 0.0, E4 0.0, E5 0.0, E6 0.0} C_DIS
LIN {E6POS: X 1196.000, Y -232.200, Z 554.000, A 0.000, B 90.000, C 0.000, E1 0.000, E2 0.0, E3 0.0, E4 0.0, E5 0.0, E6 0.0} C_DIS
LIN {E6POS: X 1196.000, Y -233.200, Z 554.000, A 0.000, B 90.000, C 0.000, E1 0.000, E2 0.0, E3 0.0, E4 0.0, E5 0.0, E6 0.0} C_DIS
LIN {E6POS: X 1196.000, Y -234.200, Z 554.000, A 0.000, B 90.000, C 0.000, E1 0.000, E2 0.0, E3 0.0, E4 0.0, E5 0.0, E6 0.0} C_DIS
LIN {E6POS: X 1196.000, Y -235.200, Z 554.000, A 0.000, B 90.000, C 0.000, E1 0.000, E2 0.0, E3 0.0, E4 0.0, E5 0.0, E6 0.0} C_DIS
LIN {E6POS: X 1196.000, Y -236.200, Z 554.000, A 0.000, B 90.000, C 0.000, E1 0.000, E2 0.0, E3 0.0, E4 0.0, E5 0.0, E6 0.0} C_DIS
LIN {E6POS: X 1196.000, Y -237.200, Z 554.000, A 0.000, B 90.000, C 0.000, E1 0.000, E2 0.0, E3 0.0, E4 0.0, E5 0.0, E6 0.0} C_DIS
LIN {E6POS: X 1196.000, Y -237.200, Z 555.000, A 0.000, B 90.000, C 0.000, E1 0.000, E2 0.0, E3 0.0, E4 0.0, E5 0.0, E6 0.0} C_DIS
LIN {E6POS: X 1197.000, Y -237.200, Z 555.000, A 0.000, B 90.000, C 0.000, E1 0.000, E2 0.0, E3 0.0, E4 0.0, E5 0.0, E6 0.0} C_DIS
LIN {E6POS: X 1198.000, Y -237.200, Z 555.000, A 0.000, B 90.000, C 0.000, E1 0.000, E2 0.0, E3 0.0, E4 0.0, E5 0.0, E6 0.0} C_DIS
LIN {E6POS: X 1199.000, Y -237.200, Z 555.000, A 0.000, B 90.000, C 0.000, E1 0.000, E2 0.0, E3 0.0, E4 0.0, E5 0.0, E6 0.0} C_DIS
LIN {E6POS: X 1200.000, Y -237.200, Z 555.000, A 0.000, B 90.000, C 0.000, E1 0.000, E2 0.0, E3 0.0, E4 0.0, E5 0.0, E6 0.0} C_DIS
LIN {E6POS: X 1201.000, Y -237.200, Z 555.000, A 0.000, B 90.000, C 0.000, E1 0.000, E2 0.0, E3 0.0, E4 0.0, E5 0.0, E6 0.0} C_DIS
LIN {E6POS: X 1201.000, Y -237.200, Z 555.000, A 0.000, B 90.000, C 0.000, E1 0.000, E2 0.0, E3 0.0, E4 0.0, E5 0.0, E6 0.0} C_DIS
LIN {E6POS: X 1201.000, Y -236.200, Z 555.000, A 0.000, B 90.000, C 0.000, E1 0.000, E2 0.0, E3 0.0, E4 0.0, E5 0.0, E6 0.0} C_DIS
LIN {E6POS: X 1201.000, Y -235.200, Z 555.000, A 0.000, B 90.000, C 0.000, E1 0.000, E2 0.0, E3 0.0, E4 0.0, E5 0.0, E6 0.0} C_DIS
LIN {E6POS: X 1201.000, Y -234.200, Z 555.000, A 0.000, B 90.000, C 0.000, E1 0.000, E2 0.0, E3 0.0, E4 0.0, E5 0.0, E6 0.0} C_DIS
LIN {E6POS: X 1201.000, Y -233.200, Z 555.000, A 0.000, B 90.000, C 0.000, E1 0.000, E2 0.0, E3 0.0, E4 0.0, E5 0.0, E6 0.0} C_DIS
LIN {E6POS: X 1201.000, Y -232.200, Z 555.000, A 0.000, B 90.000, C 0.000, E1 0.000, E2 0.0, E3 0.0, E4 0.0, E5 0.0, E6 0.0} C_DIS
LIN {E6POS: X 1201.000, Y -231.200, Z 555.000, A 0.000, B 90.000, C 0.000, E1 0.000, E2 0.0, E3 0.0, E4 0.0, E5 0.0, E6 0.0} C_DIS
LIN {E6POS: X 1201.000, Y -230.200, Z 555.000, A 0.000, B 90.000, C 0.000, E1 0.000, E2 0.0, E3 0.0, E4 0.0, E5 0.0, E6 0.0} C_DIS
LIN {E6POS: X 1201.000, Y -229.200, Z 555.000, A 0.000, B 90.000, C 0.000, E1 0.000, E2 0.0, E3 0.0, E4 0.0, E5 0.0, E6 0.0} C_DIS
LIN {E6POS: X 1201.000, Y -228.200, Z 555.000, A 0.000, B 90.000, C 0.000, E1 0.000, E2 0.0, E3 0.0, E4 0.0, E5 0.0, E6 0.0} C_DIS
LIN {E6POS: X 1201.000, Y -227.200, Z 555.000, A 0.000, B 90.000, C 0.000, E1 0.000, E2 0.0, E3 0.0, E4 0.0, E5 0.0, E6 0.0} C_DIS
LIN {E6POS: X 1201.000, Y -226.200, Z 555.000, A 0.000, B 90.000, C 0.000, E1 0.000, E2 0.0, E3 0.0, E4 0.0, E5 0.0, E6 0.0} C_DIS
LIN {E6POS: X 1201.000, Y -225.200, Z 555.000, A 0.000, B 90.000, C 0.000, E1 0.000, E2 0.0, E3 0.0, E4 0.0, E5 0.0, E6 0.0} C_DIS
LIN {E6POS: X 1201.000, Y -224.200, Z 555.000, A 0.000, B 90.000, C 0.000, E1 0.000, E2 0.0, E3 0.0, E4 0.0, E5 0.0, E6 0.0} C_DIS
LIN {E6POS: X 1201.000, Y -223.200, Z 555.000, A 0.000, B 90.000, C 0.000, E1 0.000, E2 0.0, E3 0.0, E4 0.0, E5 0.0, E6 0.0} C_DIS
LIN {E6POS: X 1201.000, Y -222.200, Z 555.000, A 0.000, B 90.000, C 0.000, E1 0.000, E2 0.0, E3 0.0, E4 0.0, E5 0.0, E6 0.0} C_DIS
LIN {E6POS: X 1201.000, Y -221.200, Z 555.000, A 0.000, B 90.000, C 0.000, E1 0.000, E2 0.0, E3 0.0, E4 0.0, E5 0.0, E6 0.0} C_DIS
LIN {E6POS: X 1201.000, Y -220.200, Z 555.000, A 0.000, B 90.000, C 0.000, E1 0.000, E2 0.0, E3 0.0, E4 0.0, E5 0.0, E6 0.0} C_DIS
LIN {E6POS: X 1201.000, Y -219.200, Z 555.000, A 0.000, B 90.000, C 0.000, E1 0.000, E2 0.0, E3 0.0, E4 0.0, E5 0.0, E6 0.0} C_DIS
LIN {E6POS: X 1201.000, Y -218.200, Z 555.000, A 0.000, B 90.000, C 0.000, E1 0.000, E2 0.0, E3 0.0, E4 0.0, E5 0.0, E6 0.0} C_DIS
LIN {E6POS: X 1201.000, Y -217.200, Z 555.000, A 0.000, B 90.000, C 0.000, E1 0.000, E2 0.0, E3 0.0, E4 0.0, E5 0.0, E6 0.0} C_DIS
LIN {E6POS: X 1201.000, Y -216.200, Z 555.000, A 0.000, B 90.000, C 0.000, E1 0.000, E2 0.0, E3 0.0, E4 0.0, E5 0.0, E6 0.0} C_DIS
LIN {E6POS: X 1201.000, Y -215.200, Z 555.000, A 0.000, B 90.000, C 0.000, E1 0.000, E2 0.0, E3 0.0, E4 0.0, E5 0.0, E6 0.0} C_DIS
LIN {E6POS: X 1201.000, Y -214.200, Z 555.000, A 0.000, B 90.000, C 0.000, E1 0.000, E2 0.0, E3 0.0, E4 0.0, E5 0.0, E6 0.0} C_DIS
LIN {E6POS: X 1201.000, Y -213.200, Z 555.000, A 0.000, B 90.000, C 0.000, E1 0.000, E2 0.0, E3 0.0, E4 0.0, E5 0.0, E6 0.0} C_DIS
LIN {E6POS: X 1201.000, Y -212.200, Z 555.000, A 0.000, B 90.000, C 0.000, E1 0.000, E2 0.0, E3 0.0, E4 0.0, E5 0.0, E6 0.0} C_DIS
LIN {E6POS: X 1201.000, Y -211.200, Z 555.000, A 0.000, B 90.000, C 0.000, E1 0.000, E2 0.0, E3 0.0, E4 0.0, E5 0.0, E6 0.0} C_DIS
LIN {E6POS: X 1201.000, Y -210.200, Z 555.000, A 0.000, B 90.000, C 0.000, E1 0.000, E2 0.0, E3 0.0, E4 0.0, E5 0.0, E6 0.0} C_DIS
LIN {E6POS: X 1201.000, Y -209.200, Z 555.000, A 0.000, B 90.000, C 0.000, E1 0.000, E2 0.0, E3 0.0, E4 0.0, E5 0.0, E6 0.0} C_DIS
LIN {E6POS: X 1201.000, Y -208.200, Z 555.000, A 0.000, B 90.000, C 0.000, E1 0.000, E2 0.0, E3 0.0, E4 0.0, E5 0.0, E6 0.0} C_DIS
LIN {E6POS: X 1201.000, Y -207.200, Z 555.000, A 0.000, B 90.000, C 0.000, E1 0.000, E2 0.0, E3 0.0, E4 0.0, E5 0.0, E6 0.0} C_DIS
LIN {E6POS: X 1201.000, Y -206.200, Z 555.000, A 0.000, B 90.000, C 0.000, E1 0.000, E2 0.0, E3 0.0, E4 0.0, E5 0.0, E6 0.0} C_DIS
LIN {E6POS: X 1201.000, Y -205.200, Z 555.000, A 0.000, B 90.000, C 0.000, E1 0.000, E2 0.0, E3 0.0, E4 0.0, E5 0.0, E6 0.0} C_DIS
LIN {E6POS: X 1201.000, Y -204.200, Z 555.000, A 0.000, B 90.000, C 0.000, E1 0.000, E2 0.0, E3 0.0, E4 0.0, E5 0.0, E6 0.0} C_DIS
LIN {E6POS: X 1201.000, Y -203.200, Z 555.000, A 0.000, B 90.000, C 0.000, E1 0.000, E2 0.0, E3 0.0, E4 0.0, E5 0.0, E6 0.0} C_DIS
LIN {E6POS: X 1201.000, Y -202.200, Z 555.000, A 0.000, B 90.000, C 0.000, E1 0.000, E2 0.0, E3 0.0, E4 0.0, E5 0.0, E6 0.0} C_DIS
LIN {E6POS: X 1201.000, Y -201.200, Z 555.000, A 0.000, B 90.000, C 0.000, E1 0.000, E2 0.0, E3 0.0, E4 0.0, E5 0.0, E6 0.0} C_DIS
LIN {E6POS: X 1201.000, Y -200.200, Z 555.000, A 0.000, B 90.000, C 0.000, E1 0.000, E2 0.0, E3 0.0, E4 0.0, E5 0.0, E6 0.0} C_DIS
LIN {E6POS: X 1201.000, Y -199.200, Z 555.000, A 0.000, B 90.000, C 0.000, E1 0.000, E2 0.0, E3 0.0, E4 0.0, E5 0.0, E6 0.0} C_DIS
LIN {E6POS: X 1201.000, Y -198.200, Z 555.000, A 0.000, B 90.000, C 0.000, E1 0.000, E2 0.0, E3 0.0, E4 0.0, E5 0.0, E6 0.0} C_DIS
LIN {E6POS: X 1201.000, Y -197.200, Z 555.000, A 0.000, B 90.000, C 0.000, E1 0.000, E2 0.0, E3 0.0, E4 0.0, E5 0.0, E6 0.0} C_DIS
LIN {E6POS: X 1201.000, Y -196.200, Z 555.000, A 0.000, B 90.000, C 0.000, E1 0.000, E2 0.0, E3 0.0, E4 0.0, E5 0.0, E6 0.0} C_DIS
LIN {E6POS: X 1201.000, Y -195.200, Z 555.000, A 0.000, B 90.000, C 0.000, E1 0.000, E2 0.0, E3 0.0, E4 0.0, E5 0.0, E6 0.0} C_DIS
LIN {E6POS: X 1201.000, Y -194.200, Z 555.000, A 0.000, B 90.000, C 0.000, E1 0.000, E2 0.0, E3 0.0, E4 0.0, E5 0.0, E6 0.0} C_DIS
LIN {E6POS: X 1201.000, Y -193.200, Z 555.000, A 0.000, B 90.000, C 0.000, E1 0.000, E2 0.0, E3 0.0, E4 0.0, E5 0.0, E6 0.0} C_DIS
LIN {E6POS: X 1201.000, Y -192.200, Z 555.000, A 0.000, B 90.000, C 0.000, E1 0.000, E2 0.0, E3 0.0, E4 0.0, E5 0.0, E6 0.0} C_DIS
LIN {E6POS: X 1201.000, Y -191.200, Z 555.000, A 0.000, B 90.000, C 0.000, E1 0.000, E2 0.0, E3 0.0, E4 0.0, E5 0.0, E6 0.0} C_DIS
LIN {E6POS: X 1201.000, Y -190.200, Z 555.000, A 0.000, B 90.000, C 0.000, E1 0.000, E2 0.0, E3 0.0, E4 0.0, E5 0.0, E6 0.0} C_DIS
LIN {E6POS: X 1201.000, Y -189.200, Z 555.000, A 0.000, B 90.000, C 0.000, E1 0.000, E2 0.0, E3 0.0, E4 0.0, E5 0.0, E6 0.0} C_DIS
LIN {E6POS: X 1201.000, Y -188.200, Z 555.000, A 0.000, B 90.000, C 0.000, E1 0.000, E2 0.0, E3 0.0, E4 0.0, E5 0.0, E6 0.0} C_DIS
LIN {E6POS: X 1201.000, Y -187.200, Z 555.000, A 0.000, B 90.000, C 0.000, E1 0.000, E2 0.0, E3 0.0, E4 0.0, E5 0.0, E6 0.0} C_DIS
LIN {E6POS: X 1201.000, Y -187.200, Z 555.000, A 0.000, B 90.000, C 0.000, E1 0.000, E2 0.0, E3 0.0, E4 0.0, E5 0.0, E6 0.0} C_DIS
LIN {E6POS: X 1200.000, Y -187.200, Z 555.000, A 0.000, B 90.000, C 0.000, E1 0.000, E2 0.0, E3 0.0, E4 0.0, E5 0.0, E6 0.0} C_DIS
LIN {E6POS: X 1199.000, Y -187.200, Z 555.000, A 0.000, B 90.000, C 0.000, E1 0.000, E2 0.0, E3 0.0, E4 0.0, E5 0.0, E6 0.0} C_DIS
LIN {E6POS: X 1198.000, Y -187.200, Z 555.000, A 0.000, B 90.000, C 0.000, E1 0.000, E2 0.0, E3 0.0, E4 0.0, E5 0.0, E6 0.0} C_DIS
LIN {E6POS: X 1197.000, Y -187.200, Z 555.000, A 0.000, B 90.000, C 0.000, E1 0.000, E2 0.0, E3 0.0, E4 0.0, E5 0.0, E6 0.0} C_DIS
LIN {E6POS: X 1196.000, Y -187.200, Z 555.000, A 0.000, B 90.000, C 0.000, E1 0.000, E2 0.0, E3 0.0, E4 0.0, E5 0.0, E6 0.0} C_DIS
LIN {E6POS: X 1196.000, Y -187.200, Z 555.000, A 0.000, B 90.000, C 0.000, E1 0.000, E2 0.0, E3 0.0, E4 0.0, E5 0.0, E6 0.0} C_DIS
LIN {E6POS: X 1196.000, Y -188.200, Z 555.000, A 0.000, B 90.000, C 0.000, E1 0.000, E2 0.0, E3 0.0, E4 0.0, E5 0.0, E6 0.0} C_DIS
LIN {E6POS: X 1196.000, Y -189.200, Z 555.000, A 0.000, B 90.000, C 0.000, E1 0.000, E2 0.0, E3 0.0, E4 0.0, E5 0.0, E6 0.0} C_DIS
LIN {E6POS: X 1196.000, Y -190.200, Z 555.000, A 0.000, B 90.000, C 0.000, E1 0.000, E2 0.0, E3 0.0, E4 0.0, E5 0.0, E6 0.0} C_DIS
LIN {E6POS: X 1196.000, Y -191.200, Z 555.000, A 0.000, B 90.000, C 0.000, E1 0.000, E2 0.0, E3 0.0, E4 0.0, E5 0.0, E6 0.0} C_DIS
LIN {E6POS: X 1196.000, Y -192.200, Z 555.000, A 0.000, B 90.000, C 0.000, E1 0.000, E2 0.0, E3 0.0, E4 0.0, E5 0.0, E6 0.0} C_DIS
LIN {E6POS: X 1196.000, Y -193.200, Z 555.000, A 0.000, B 90.000, C 0.000, E1 0.000, E2 0.0, E3 0.0, E4 0.0, E5 0.0, E6 0.0} C_DIS
LIN {E6POS: X 1196.000, Y -194.200, Z 555.000, A 0.000, B 90.000, C 0.000, E1 0.000, E2 0.0, E3 0.0, E4 0.0, E5 0.0, E6 0.0} C_DIS
LIN {E6POS: X 1196.000, Y -195.200, Z 555.000, A 0.000, B 90.000, C 0.000, E1 0.000, E2 0.0, E3 0.0, E4 0.0, E5 0.0, E6 0.0} C_DIS
LIN {E6POS: X 1196.000, Y -196.200, Z 555.000, A 0.000, B 90.000, C 0.000, E1 0.000, E2 0.0, E3 0.0, E4 0.0, E5 0.0, E6 0.0} C_DIS
LIN {E6POS: X 1196.000, Y -197.200, Z 555.000, A 0.000, B 90.000, C 0.000, E1 0.000, E2 0.0, E3 0.0, E4 0.0, E5 0.0, E6 0.0} C_DIS
LIN {E6POS: X 1196.000, Y -198.200, Z 555.000, A 0.000, B 90.000, C 0.000, E1 0.000, E2 0.0, E3 0.0, E4 0.0, E5 0.0, E6 0.0} C_DIS
LIN {E6POS: X 1196.000, Y -199.200, Z 555.000, A 0.000, B 90.000, C 0.000, E1 0.000, E2 0.0, E3 0.0, E4 0.0, E5 0.0, E6 0.0} C_DIS
LIN {E6POS: X 1196.000, Y -200.200, Z 555.000, A 0.000, B 90.000, C 0.000, E1 0.000, E2 0.0, E3 0.0, E4 0.0, E5 0.0, E6 0.0} C_DIS
LIN {E6POS: X 1196.000, Y -201.200, Z 555.000, A 0.000, B 90.000, C 0.000, E1 0.000, E2 0.0, E3 0.0, E4 0.0, E5 0.0, E6 0.0} C_DIS
LIN {E6POS: X 1196.000, Y -202.200, Z 555.000, A 0.000, B 90.000, C 0.000, E1 0.000, E2 0.0, E3 0.0, E4 0.0, E5 0.0, E6 0.0} C_DIS
LIN {E6POS: X 1196.000, Y -203.200, Z 555.000, A 0.000, B 90.000, C 0.000, E1 0.000, E2 0.0, E3 0.0, E4 0.0, E5 0.0, E6 0.0} C_DIS
LIN {E6POS: X 1196.000, Y -204.200, Z 555.000, A 0.000, B 90.000, C 0.000, E1 0.000, E2 0.0, E3 0.0, E4 0.0, E5 0.0, E6 0.0} C_DIS
LIN {E6POS: X 1196.000, Y -205.200, Z 555.000, A 0.000, B 90.000, C 0.000, E1 0.000, E2 0.0, E3 0.0, E4 0.0, E5 0.0, E6 0.0} C_DIS
LIN {E6POS: X 1196.000, Y -206.200, Z 555.000, A 0.000, B 90.000, C 0.000, E1 0.000, E2 0.0, E3 0.0, E4 0.0, E5 0.0, E6 0.0} C_DIS
LIN {E6POS: X 1196.000, Y -207.200, Z 555.000, A 0.000, B 90.000, C 0.000, E1 0.000, E2 0.0, E3 0.0, E4 0.0, E5 0.0, E6 0.0} C_DIS
LIN {E6POS: X 1196.000, Y -208.200, Z 555.000, A 0.000, B 90.000, C 0.000, E1 0.000, E2 0.0, E3 0.0, E4 0.0, E5 0.0, E6 0.0} C_DIS
LIN {E6POS: X 1196.000, Y -209.200, Z 555.000, A 0.000, B 90.000, C 0.000, E1 0.000, E2 0.0, E3 0.0, E4 0.0, E5 0.0, E6 0.0} C_DIS
LIN {E6POS: X 1196.000, Y -210.200, Z 555.000, A 0.000, B 90.000, C 0.000, E1 0.000, E2 0.0, E3 0.0, E4 0.0, E5 0.0, E6 0.0} C_DIS
LIN {E6POS: X 1196.000, Y -211.200, Z 555.000, A 0.000, B 90.000, C 0.000, E1 0.000, E2 0.0, E3 0.0, E4 0.0, E5 0.0, E6 0.0} C_DIS
LIN {E6POS: X 1196.000, Y -212.200, Z 555.000, A 0.000, B 90.000, C 0.000, E1 0.000, E2 0.0, E3 0.0, E4 0.0, E5 0.0, E6 0.0} C_DIS
LIN {E6POS: X 1196.000, Y -213.200, Z 555.000, A 0.000, B 90.000, C 0.000, E1 0.000, E2 0.0, E3 0.0, E4 0.0, E5 0.0, E6 0.0} C_DIS
LIN {E6POS: X 1196.000, Y -214.200, Z 555.000, A 0.000, B 90.000, C 0.000, E1 0.000, E2 0.0, E3 0.0, E4 0.0, E5 0.0, E6 0.0} C_DIS
LIN {E6POS: X 1196.000, Y -215.200, Z 555.000, A 0.000, B 90.000, C 0.000, E1 0.000, E2 0.0, E3 0.0, E4 0.0, E5 0.0, E6 0.0} C_DIS
LIN {E6POS: X 1196.000, Y -216.200, Z 555.000, A 0.000, B 90.000, C 0.000, E1 0.000, E2 0.0, E3 0.0, E4 0.0, E5 0.0, E6 0.0} C_DIS
LIN {E6POS: X 1196.000, Y -217.200, Z 555.000, A 0.000, B 90.000, C 0.000, E1 0.000, E2 0.0, E3 0.0, E4 0.0, E5 0.0, E6 0.0} C_DIS
LIN {E6POS: X 1196.000, Y -218.200, Z 555.000, A 0.000, B 90.000, C 0.000, E1 0.000, E2 0.0, E3 0.0, E4 0.0, E5 0.0, E6 0.0} C_DIS
LIN {E6POS: X 1196.000, Y -219.200, Z 555.000, A 0.000, B 90.000, C 0.000, E1 0.000, E2 0.0, E3 0.0, E4 0.0, E5 0.0, E6 0.0} C_DIS
LIN {E6POS: X 1196.000, Y -220.200, Z 555.000, A 0.000, B 90.000, C 0.000, E1 0.000, E2 0.0, E3 0.0, E4 0.0, E5 0.0, E6 0.0} C_DIS
LIN {E6POS: X 1196.000, Y -221.200, Z 555.000, A 0.000, B 90.000, C 0.000, E1 0.000, E2 0.0, E3 0.0, E4 0.0, E5 0.0, E6 0.0} C_DIS
LIN {E6POS: X 1196.000, Y -222.200, Z 555.000, A 0.000, B 90.000, C 0.000, E1 0.000, E2 0.0, E3 0.0, E4 0.0, E5 0.0, E6 0.0} C_DIS
LIN {E6POS: X 1196.000, Y -223.200, Z 555.000, A 0.000, B 90.000, C 0.000, E1 0.000, E2 0.0, E3 0.0, E4 0.0, E5 0.0, E6 0.0} C_DIS
LIN {E6POS: X 1196.000, Y -224.200, Z 555.000, A 0.000, B 90.000, C 0.000, E1 0.000, E2 0.0, E3 0.0, E4 0.0, E5 0.0, E6 0.0} C_DIS
LIN {E6POS: X 1196.000, Y -225.200, Z 555.000, A 0.000, B 90.000, C 0.000, E1 0.000, E2 0.0, E3 0.0, E4 0.0, E5 0.0, E6 0.0} C_DIS
LIN {E6POS: X 1196.000, Y -226.200, Z 555.000, A 0.000, B 90.000, C 0.000, E1 0.000, E2 0.0, E3 0.0, E4 0.0, E5 0.0, E6 0.0} C_DIS
LIN {E6POS: X 1196.000, Y -227.200, Z 555.000, A 0.000, B 90.000, C 0.000, E1 0.000, E2 0.0, E3 0.0, E4 0.0, E5 0.0, E6 0.0} C_DIS
LIN {E6POS: X 1196.000, Y -228.200, Z 555.000, A 0.000, B 90.000, C 0.000, E1 0.000, E2 0.0, E3 0.0, E4 0.0, E5 0.0, E6 0.0} C_DIS
LIN {E6POS: X 1196.000, Y -229.200, Z 555.000, A 0.000, B 90.000, C 0.000, E1 0.000, E2 0.0, E3 0.0, E4 0.0, E5 0.0, E6 0.0} C_DIS
LIN {E6POS: X 1196.000, Y -230.200, Z 555.000, A 0.000, B 90.000, C 0.000, E1 0.000, E2 0.0, E3 0.0, E4 0.0, E5 0.0, E6 0.0} C_DIS
LIN {E6POS: X 1196.000, Y -231.200, Z 555.000, A 0.000, B 90.000, C 0.000, E1 0.000, E2 0.0, E3 0.0, E4 0.0, E5 0.0, E6 0.0} C_DIS
LIN {E6POS: X 1196.000, Y -232.200, Z 555.000, A 0.000, B 90.000, C 0.000, E1 0.000, E2 0.0, E3 0.0, E4 0.0, E5 0.0, E6 0.0} C_DIS
LIN {E6POS: X 1196.000, Y -233.200, Z 555.000, A 0.000, B 90.000, C 0.000, E1 0.000, E2 0.0, E3 0.0, E4 0.0, E5 0.0, E6 0.0} C_DIS
LIN {E6POS: X 1196.000, Y -234.200, Z 555.000, A 0.000, B 90.000, C 0.000, E1 0.000, E2 0.0, E3 0.0, E4 0.0, E5 0.0, E6 0.0} C_DIS
LIN {E6POS: X 1196.000, Y -235.200, Z 555.000, A 0.000, B 90.000, C 0.000, E1 0.000, E2 0.0, E3 0.0, E4 0.0, E5 0.0, E6 0.0} C_DIS
LIN {E6POS: X 1196.000, Y -236.200, Z 555.000, A 0.000, B 90.000, C 0.000, E1 0.000, E2 0.0, E3 0.0, E4 0.0, E5 0.0, E6 0.0} C_DIS
LIN {E6POS: X 1196.000, Y -237.200, Z 555.000, A 0.000, B 90.000, C 0.000, E1 0.000, E2 0.0, E3 0.0, E4 0.0, E5 0.0, E6 0.0} C_DIS
LIN {E6POS: X 1196.000, Y -237.200, Z 556.000, A 0.000, B 90.000, C 0.000, E1 0.000, E2 0.0, E3 0.0, E4 0.0, E5 0.0, E6 0.0} C_DIS
LIN {E6POS: X 1197.000, Y -237.200, Z 556.000, A 0.000, B 90.000, C 0.000, E1 0.000, E2 0.0, E3 0.0, E4 0.0, E5 0.0, E6 0.0} C_DIS
LIN {E6POS: X 1198.000, Y -237.200, Z 556.000, A 0.000, B 90.000, C 0.000, E1 0.000, E2 0.0, E3 0.0, E4 0.0, E5 0.0, E6 0.0} C_DIS
LIN {E6POS: X 1199.000, Y -237.200, Z 556.000, A 0.000, B 90.000, C 0.000, E1 0.000, E2 0.0, E3 0.0, E4 0.0, E5 0.0, E6 0.0} C_DIS
LIN {E6POS: X 1200.000, Y -237.200, Z 556.000, A 0.000, B 90.000, C 0.000, E1 0.000, E2 0.0, E3 0.0, E4 0.0, E5 0.0, E6 0.0} C_DIS
LIN {E6POS: X 1201.000, Y -237.200, Z 556.000, A 0.000, B 90.000, C 0.000, E1 0.000, E2 0.0, E3 0.0, E4 0.0, E5 0.0, E6 0.0} C_DIS
LIN {E6POS: X 1201.000, Y -237.200, Z 556.000, A 0.000, B 90.000, C 0.000, E1 0.000, E2 0.0, E3 0.0, E4 0.0, E5 0.0, E6 0.0} C_DIS
LIN {E6POS: X 1201.000, Y -236.200, Z 556.000, A 0.000, B 90.000, C 0.000, E1 0.000, E2 0.0, E3 0.0, E4 0.0, E5 0.0, E6 0.0} C_DIS
LIN {E6POS: X 1201.000, Y -235.200, Z 556.000, A 0.000, B 90.000, C 0.000, E1 0.000, E2 0.0, E3 0.0, E4 0.0, E5 0.0, E6 0.0} C_DIS
LIN {E6POS: X 1201.000, Y -234.200, Z 556.000, A 0.000, B 90.000, C 0.000, E1 0.000, E2 0.0, E3 0.0, E4 0.0, E5 0.0, E6 0.0} C_DIS
LIN {E6POS: X 1201.000, Y -233.200, Z 556.000, A 0.000, B 90.000, C 0.000, E1 0.000, E2 0.0, E3 0.0, E4 0.0, E5 0.0, E6 0.0} C_DIS
LIN {E6POS: X 1201.000, Y -232.200, Z 556.000, A 0.000, B 90.000, C 0.000, E1 0.000, E2 0.0, E3 0.0, E4 0.0, E5 0.0, E6 0.0} C_DIS
LIN {E6POS: X 1201.000, Y -231.200, Z 556.000, A 0.000, B 90.000, C 0.000, E1 0.000, E2 0.0, E3 0.0, E4 0.0, E5 0.0, E6 0.0} C_DIS
LIN {E6POS: X 1201.000, Y -230.200, Z 556.000, A 0.000, B 90.000, C 0.000, E1 0.000, E2 0.0, E3 0.0, E4 0.0, E5 0.0, E6 0.0} C_DIS
LIN {E6POS: X 1201.000, Y -229.200, Z 556.000, A 0.000, B 90.000, C 0.000, E1 0.000, E2 0.0, E3 0.0, E4 0.0, E5 0.0, E6 0.0} C_DIS
LIN {E6POS: X 1201.000, Y -228.200, Z 556.000, A 0.000, B 90.000, C 0.000, E1 0.000, E2 0.0, E3 0.0, E4 0.0, E5 0.0, E6 0.0} C_DIS
LIN {E6POS: X 1201.000, Y -227.200, Z 556.000, A 0.000, B 90.000, C 0.000, E1 0.000, E2 0.0, E3 0.0, E4 0.0, E5 0.0, E6 0.0} C_DIS
LIN {E6POS: X 1201.000, Y -226.200, Z 556.000, A 0.000, B 90.000, C 0.000, E1 0.000, E2 0.0, E3 0.0, E4 0.0, E5 0.0, E6 0.0} C_DIS
LIN {E6POS: X 1201.000, Y -225.200, Z 556.000, A 0.000, B 90.000, C 0.000, E1 0.000, E2 0.0, E3 0.0, E4 0.0, E5 0.0, E6 0.0} C_DIS
LIN {E6POS: X 1201.000, Y -224.200, Z 556.000, A 0.000, B 90.000, C 0.000, E1 0.000, E2 0.0, E3 0.0, E4 0.0, E5 0.0, E6 0.0} C_DIS
LIN {E6POS: X 1201.000, Y -223.200, Z 556.000, A 0.000, B 90.000, C 0.000, E1 0.000, E2 0.0, E3 0.0, E4 0.0, E5 0.0, E6 0.0} C_DIS
LIN {E6POS: X 1201.000, Y -222.200, Z 556.000, A 0.000, B 90.000, C 0.000, E1 0.000, E2 0.0, E3 0.0, E4 0.0, E5 0.0, E6 0.0} C_DIS
LIN {E6POS: X 1201.000, Y -221.200, Z 556.000, A 0.000, B 90.000, C 0.000, E1 0.000, E2 0.0, E3 0.0, E4 0.0, E5 0.0, E6 0.0} C_DIS
LIN {E6POS: X 1201.000, Y -220.200, Z 556.000, A 0.000, B 90.000, C 0.000, E1 0.000, E2 0.0, E3 0.0, E4 0.0, E5 0.0, E6 0.0} C_DIS
LIN {E6POS: X 1201.000, Y -219.200, Z 556.000, A 0.000, B 90.000, C 0.000, E1 0.000, E2 0.0, E3 0.0, E4 0.0, E5 0.0, E6 0.0} C_DIS
LIN {E6POS: X 1201.000, Y -218.200, Z 556.000, A 0.000, B 90.000, C 0.000, E1 0.000, E2 0.0, E3 0.0, E4 0.0, E5 0.0, E6 0.0} C_DIS
LIN {E6POS: X 1201.000, Y -217.200, Z 556.000, A 0.000, B 90.000, C 0.000, E1 0.000, E2 0.0, E3 0.0, E4 0.0, E5 0.0, E6 0.0} C_DIS
LIN {E6POS: X 1201.000, Y -216.200, Z 556.000, A 0.000, B 90.000, C 0.000, E1 0.000, E2 0.0, E3 0.0, E4 0.0, E5 0.0, E6 0.0} C_DIS
LIN {E6POS: X 1201.000, Y -215.200, Z 556.000, A 0.000, B 90.000, C 0.000, E1 0.000, E2 0.0, E3 0.0, E4 0.0, E5 0.0, E6 0.0} C_DIS
LIN {E6POS: X 1201.000, Y -214.200, Z 556.000, A 0.000, B 90.000, C 0.000, E1 0.000, E2 0.0, E3 0.0, E4 0.0, E5 0.0, E6 0.0} C_DIS
LIN {E6POS: X 1201.000, Y -213.200, Z 556.000, A 0.000, B 90.000, C 0.000, E1 0.000, E2 0.0, E3 0.0, E4 0.0, E5 0.0, E6 0.0} C_DIS
LIN {E6POS: X 1201.000, Y -212.200, Z 556.000, A 0.000, B 90.000, C 0.000, E1 0.000, E2 0.0, E3 0.0, E4 0.0, E5 0.0, E6 0.0} C_DIS
LIN {E6POS: X 1201.000, Y -211.200, Z 556.000, A 0.000, B 90.000, C 0.000, E1 0.000, E2 0.0, E3 0.0, E4 0.0, E5 0.0, E6 0.0} C_DIS
LIN {E6POS: X 1201.000, Y -210.200, Z 556.000, A 0.000, B 90.000, C 0.000, E1 0.000, E2 0.0, E3 0.0, E4 0.0, E5 0.0, E6 0.0} C_DIS
LIN {E6POS: X 1201.000, Y -209.200, Z 556.000, A 0.000, B 90.000, C 0.000, E1 0.000, E2 0.0, E3 0.0, E4 0.0, E5 0.0, E6 0.0} C_DIS
LIN {E6POS: X 1201.000, Y -208.200, Z 556.000, A 0.000, B 90.000, C 0.000, E1 0.000, E2 0.0, E3 0.0, E4 0.0, E5 0.0, E6 0.0} C_DIS
LIN {E6POS: X 1201.000, Y -207.200, Z 556.000, A 0.000, B 90.000, C 0.000, E1 0.000, E2 0.0, E3 0.0, E4 0.0, E5 0.0, E6 0.0} C_DIS
LIN {E6POS: X 1201.000, Y -206.200, Z 556.000, A 0.000, B 90.000, C 0.000, E1 0.000, E2 0.0, E3 0.0, E4 0.0, E5 0.0, E6 0.0} C_DIS
LIN {E6POS: X 1201.000, Y -205.200, Z 556.000, A 0.000, B 90.000, C 0.000, E1 0.000, E2 0.0, E3 0.0, E4 0.0, E5 0.0, E6 0.0} C_DIS
LIN {E6POS: X 1201.000, Y -204.200, Z 556.000, A 0.000, B 90.000, C 0.000, E1 0.000, E2 0.0, E3 0.0, E4 0.0, E5 0.0, E6 0.0} C_DIS
LIN {E6POS: X 1201.000, Y -203.200, Z 556.000, A 0.000, B 90.000, C 0.000, E1 0.000, E2 0.0, E3 0.0, E4 0.0, E5 0.0, E6 0.0} C_DIS
LIN {E6POS: X 1201.000, Y -202.200, Z 556.000, A 0.000, B 90.000, C 0.000, E1 0.000, E2 0.0, E3 0.0, E4 0.0, E5 0.0, E6 0.0} C_DIS
LIN {E6POS: X 1201.000, Y -201.200, Z 556.000, A 0.000, B 90.000, C 0.000, E1 0.000, E2 0.0, E3 0.0, E4 0.0, E5 0.0, E6 0.0} C_DIS
LIN {E6POS: X 1201.000, Y -200.200, Z 556.000, A 0.000, B 90.000, C 0.000, E1 0.000, E2 0.0, E3 0.0, E4 0.0, E5 0.0, E6 0.0} C_DIS
LIN {E6POS: X 1201.000, Y -199.200, Z 556.000, A 0.000, B 90.000, C 0.000, E1 0.000, E2 0.0, E3 0.0, E4 0.0, E5 0.0, E6 0.0} C_DIS
LIN {E6POS: X 1201.000, Y -198.200, Z 556.000, A 0.000, B 90.000, C 0.000, E1 0.000, E2 0.0, E3 0.0, E4 0.0, E5 0.0, E6 0.0} C_DIS
LIN {E6POS: X 1201.000, Y -197.200, Z 556.000, A 0.000, B 90.000, C 0.000, E1 0.000, E2 0.0, E3 0.0, E4 0.0, E5 0.0, E6 0.0} C_DIS
LIN {E6POS: X 1201.000, Y -196.200, Z 556.000, A 0.000, B 90.000, C 0.000, E1 0.000, E2 0.0, E3 0.0, E4 0.0, E5 0.0, E6 0.0} C_DIS
LIN {E6POS: X 1201.000, Y -195.200, Z 556.000, A 0.000, B 90.000, C 0.000, E1 0.000, E2 0.0, E3 0.0, E4 0.0, E5 0.0, E6 0.0} C_DIS
LIN {E6POS: X 1201.000, Y -194.200, Z 556.000, A 0.000, B 90.000, C 0.000, E1 0.000, E2 0.0, E3 0.0, E4 0.0, E5 0.0, E6 0.0} C_DIS
LIN {E6POS: X 1201.000, Y -193.200, Z 556.000, A 0.000, B 90.000, C 0.000, E1 0.000, E2 0.0, E3 0.0, E4 0.0, E5 0.0, E6 0.0} C_DIS
LIN {E6POS: X 1201.000, Y -192.200, Z 556.000, A 0.000, B 90.000, C 0.000, E1 0.000, E2 0.0, E3 0.0, E4 0.0, E5 0.0, E6 0.0} C_DIS
LIN {E6POS: X 1201.000, Y -191.200, Z 556.000, A 0.000, B 90.000, C 0.000, E1 0.000, E2 0.0, E3 0.0, E4 0.0, E5 0.0, E6 0.0} C_DIS
LIN {E6POS: X 1201.000, Y -190.200, Z 556.000, A 0.000, B 90.000, C 0.000, E1 0.000, E2 0.0, E3 0.0, E4 0.0, E5 0.0, E6 0.0} C_DIS
LIN {E6POS: X 1201.000, Y -189.200, Z 556.000, A 0.000, B 90.000, C 0.000, E1 0.000, E2 0.0, E3 0.0, E4 0.0, E5 0.0, E6 0.0} C_DIS
LIN {E6POS: X 1201.000, Y -188.200, Z 556.000, A 0.000, B 90.000, C 0.000, E1 0.000, E2 0.0, E3 0.0, E4 0.0, E5 0.0, E6 0.0} C_DIS
LIN {E6POS: X 1201.000, Y -187.200, Z 556.000, A 0.000, B 90.000, C 0.000, E1 0.000, E2 0.0, E3 0.0, E4 0.0, E5 0.0, E6 0.0} C_DIS
LIN {E6POS: X 1201.000, Y -187.200, Z 556.000, A 0.000, B 90.000, C 0.000, E1 0.000, E2 0.0, E3 0.0, E4 0.0, E5 0.0, E6 0.0} C_DIS
LIN {E6POS: X 1200.000, Y -187.200, Z 556.000, A 0.000, B 90.000, C 0.000, E1 0.000, E2 0.0, E3 0.0, E4 0.0, E5 0.0, E6 0.0} C_DIS
LIN {E6POS: X 1199.000, Y -187.200, Z 556.000, A 0.000, B 90.000, C 0.000, E1 0.000, E2 0.0, E3 0.0, E4 0.0, E5 0.0, E6 0.0} C_DIS
LIN {E6POS: X 1198.000, Y -187.200, Z 556.000, A 0.000, B 90.000, C 0.000, E1 0.000, E2 0.0, E3 0.0, E4 0.0, E5 0.0, E6 0.0} C_DIS
LIN {E6POS: X 1197.000, Y -187.200, Z 556.000, A 0.000, B 90.000, C 0.000, E1 0.000, E2 0.0, E3 0.0, E4 0.0, E5 0.0, E6 0.0} C_DIS
LIN {E6POS: X 1196.000, Y -187.200, Z 556.000, A 0.000, B 90.000, C 0.000, E1 0.000, E2 0.0, E3 0.0, E4 0.0, E5 0.0, E6 0.0} C_DIS
LIN {E6POS: X 1196.000, Y -187.200, Z 556.000, A 0.000, B 90.000, C 0.000, E1 0.000, E2 0.0, E3 0.0, E4 0.0, E5 0.0, E6 0.0} C_DIS
LIN {E6POS: X 1196.000, Y -188.200, Z 556.000, A 0.000, B 90.000, C 0.000, E1 0.000, E2 0.0, E3 0.0, E4 0.0, E5 0.0, E6 0.0} C_DIS
LIN {E6POS: X 1196.000, Y -189.200, Z 556.000, A 0.000, B 90.000, C 0.000, E1 0.000, E2 0.0, E3 0.0, E4 0.0, E5 0.0, E6 0.0} C_DIS
LIN {E6POS: X 1196.000, Y -190.200, Z 556.000, A 0.000, B 90.000, C 0.000, E1 0.000, E2 0.0, E3 0.0, E4 0.0, E5 0.0, E6 0.0} C_DIS
LIN {E6POS: X 1196.000, Y -191.200, Z 556.000, A 0.000, B 90.000, C 0.000, E1 0.000, E2 0.0, E3 0.0, E4 0.0, E5 0.0, E6 0.0} C_DIS
LIN {E6POS: X 1196.000, Y -192.200, Z 556.000, A 0.000, B 90.000, C 0.000, E1 0.000, E2 0.0, E3 0.0, E4 0.0, E5 0.0, E6 0.0} C_DIS
LIN {E6POS: X 1196.000, Y -193.200, Z 556.000, A 0.000, B 90.000, C 0.000, E1 0.000, E2 0.0, E3 0.0, E4 0.0, E5 0.0, E6 0.0} C_DIS
LIN {E6POS: X 1196.000, Y -194.200, Z 556.000, A 0.000, B 90.000, C 0.000, E1 0.000, E2 0.0, E3 0.0, E4 0.0, E5 0.0, E6 0.0} C_DIS
LIN {E6POS: X 1196.000, Y -195.200, Z 556.000, A 0.000, B 90.000, C 0.000, E1 0.000, E2 0.0, E3 0.0, E4 0.0, E5 0.0, E6 0.0} C_DIS
LIN {E6POS: X 1196.000, Y -196.200, Z 556.000, A 0.000, B 90.000, C 0.000, E1 0.000, E2 0.0, E3 0.0, E4 0.0, E5 0.0, E6 0.0} C_DIS
LIN {E6POS: X 1196.000, Y -197.200, Z 556.000, A 0.000, B 90.000, C 0.000, E1 0.000, E2 0.0, E3 0.0, E4 0.0, E5 0.0, E6 0.0} C_DIS
LIN {E6POS: X 1196.000, Y -198.200, Z 556.000, A 0.000, B 90.000, C 0.000, E1 0.000, E2 0.0, E3 0.0, E4 0.0, E5 0.0, E6 0.0} C_DIS
LIN {E6POS: X 1196.000, Y -199.200, Z 556.000, A 0.000, B 90.000, C 0.000, E1 0.000, E2 0.0, E3 0.0, E4 0.0, E5 0.0, E6 0.0} C_DIS
LIN {E6POS: X 1196.000, Y -200.200, Z 556.000, A 0.000, B 90.000, C 0.000, E1 0.000, E2 0.0, E3 0.0, E4 0.0, E5 0.0, E6 0.0} C_DIS
LIN {E6POS: X 1196.000, Y -201.200, Z 556.000, A 0.000, B 90.000, C 0.000, E1 0.000, E2 0.0, E3 0.0, E4 0.0, E5 0.0, E6 0.0} C_DIS
LIN {E6POS: X 1196.000, Y -202.200, Z 556.000, A 0.000, B 90.000, C 0.000, E1 0.000, E2 0.0, E3 0.0, E4 0.0, E5 0.0, E6 0.0} C_DIS
LIN {E6POS: X 1196.000, Y -203.200, Z 556.000, A 0.000, B 90.000, C 0.000, E1 0.000, E2 0.0, E3 0.0, E4 0.0, E5 0.0, E6 0.0} C_DIS
LIN {E6POS: X 1196.000, Y -204.200, Z 556.000, A 0.000, B 90.000, C 0.000, E1 0.000, E2 0.0, E3 0.0, E4 0.0, E5 0.0, E6 0.0} C_DIS
LIN {E6POS: X 1196.000, Y -205.200, Z 556.000, A 0.000, B 90.000, C 0.000, E1 0.000, E2 0.0, E3 0.0, E4 0.0, E5 0.0, E6 0.0} C_DIS
LIN {E6POS: X 1196.000, Y -206.200, Z 556.000, A 0.000, B 90.000, C 0.000, E1 0.000, E2 0.0, E3 0.0, E4 0.0, E5 0.0, E6 0.0} C_DIS
LIN {E6POS: X 1196.000, Y -207.200, Z 556.000, A 0.000, B 90.000, C 0.000, E1 0.000, E2 0.0, E3 0.0, E4 0.0, E5 0.0, E6 0.0} C_DIS
LIN {E6POS: X 1196.000, Y -208.200, Z 556.000, A 0.000, B 90.000, C 0.000, E1 0.000, E2 0.0, E3 0.0, E4 0.0, E5 0.0, E6 0.0} C_DIS
LIN {E6POS: X 1196.000, Y -209.200, Z 556.000, A 0.000, B 90.000, C 0.000, E1 0.000, E2 0.0, E3 0.0, E4 0.0, E5 0.0, E6 0.0} C_DIS
LIN {E6POS: X 1196.000, Y -210.200, Z 556.000, A 0.000, B 90.000, C 0.000, E1 0.000, E2 0.0, E3 0.0, E4 0.0, E5 0.0, E6 0.0} C_DIS
LIN {E6POS: X 1196.000, Y -211.200, Z 556.000, A 0.000, B 90.000, C 0.000, E1 0.000, E2 0.0, E3 0.0, E4 0.0, E5 0.0, E6 0.0} C_DIS
LIN {E6POS: X 1196.000, Y -212.200, Z 556.000, A 0.000, B 90.000, C 0.000, E1 0.000, E2 0.0, E3 0.0, E4 0.0, E5 0.0, E6 0.0} C_DIS
LIN {E6POS: X 1196.000, Y -213.200, Z 556.000, A 0.000, B 90.000, C 0.000, E1 0.000, E2 0.0, E3 0.0, E4 0.0, E5 0.0, E6 0.0} C_DIS
LIN {E6POS: X 1196.000, Y -214.200, Z 556.000, A 0.000, B 90.000, C 0.000, E1 0.000, E2 0.0, E3 0.0, E4 0.0, E5 0.0, E6 0.0} C_DIS
LIN {E6POS: X 1196.000, Y -215.200, Z 556.000, A 0.000, B 90.000, C 0.000, E1 0.000, E2 0.0, E3 0.0, E4 0.0, E5 0.0, E6 0.0} C_DIS
LIN {E6POS: X 1196.000, Y -216.200, Z 556.000, A 0.000, B 90.000, C 0.000, E1 0.000, E2 0.0, E3 0.0, E4 0.0, E5 0.0, E6 0.0} C_DIS
LIN {E6POS: X 1196.000, Y -217.200, Z 556.000, A 0.000, B 90.000, C 0.000, E1 0.000, E2 0.0, E3 0.0, E4 0.0, E5 0.0, E6 0.0} C_DIS
LIN {E6POS: X 1196.000, Y -218.200, Z 556.000, A 0.000, B 90.000, C 0.000, E1 0.000, E2 0.0, E3 0.0, E4 0.0, E5 0.0, E6 0.0} C_DIS
LIN {E6POS: X 1196.000, Y -219.200, Z 556.000, A 0.000, B 90.000, C 0.000, E1 0.000, E2 0.0, E3 0.0, E4 0.0, E5 0.0, E6 0.0} C_DIS
LIN {E6POS: X 1196.000, Y -220.200, Z 556.000, A 0.000, B 90.000, C 0.000, E1 0.000, E2 0.0, E3 0.0, E4 0.0, E5 0.0, E6 0.0} C_DIS
LIN {E6POS: X 1196.000, Y -221.200, Z 556.000, A 0.000, B 90.000, C 0.000, E1 0.000, E2 0.0, E3 0.0, E4 0.0, E5 0.0, E6 0.0} C_DIS
LIN {E6POS: X 1196.000, Y -222.200, Z 556.000, A 0.000, B 90.000, C 0.000, E1 0.000, E2 0.0, E3 0.0, E4 0.0, E5 0.0, E6 0.0} C_DIS
LIN {E6POS: X 1196.000, Y -223.200, Z 556.000, A 0.000, B 90.000, C 0.000, E1 0.000, E2 0.0, E3 0.0, E4 0.0, E5 0.0, E6 0.0} C_DIS
LIN {E6POS: X 1196.000, Y -224.200, Z 556.000, A 0.000, B 90.000, C 0.000, E1 0.000, E2 0.0, E3 0.0, E4 0.0, E5 0.0, E6 0.0} C_DIS
LIN {E6POS: X 1196.000, Y -225.200, Z 556.000, A 0.000, B 90.000, C 0.000, E1 0.000, E2 0.0, E3 0.0, E4 0.0, E5 0.0, E6 0.0} C_DIS
LIN {E6POS: X 1196.000, Y -226.200, Z 556.000, A 0.000, B 90.000, C 0.000, E1 0.000, E2 0.0, E3 0.0, E4 0.0, E5 0.0, E6 0.0} C_DIS
LIN {E6POS: X 1196.000, Y -227.200, Z 556.000, A 0.000, B 90.000, C 0.000, E1 0.000, E2 0.0, E3 0.0, E4 0.0, E5 0.0, E6 0.0} C_DIS
LIN {E6POS: X 1196.000, Y -228.200, Z 556.000, A 0.000, B 90.000, C 0.000, E1 0.000, E2 0.0, E3 0.0, E4 0.0, E5 0.0, E6 0.0} C_DIS
LIN {E6POS: X 1196.000, Y -229.200, Z 556.000, A 0.000, B 90.000, C 0.000, E1 0.000, E2 0.0, E3 0.0, E4 0.0, E5 0.0, E6 0.0} C_DIS
LIN {E6POS: X 1196.000, Y -230.200, Z 556.000, A 0.000, B 90.000, C 0.000, E1 0.000, E2 0.0, E3 0.0, E4 0.0, E5 0.0, E6 0.0} C_DIS
LIN {E6POS: X 1196.000, Y -231.200, Z 556.000, A 0.000, B 90.000, C 0.000, E1 0.000, E2 0.0, E3 0.0, E4 0.0, E5 0.0, E6 0.0} C_DIS
LIN {E6POS: X 1196.000, Y -232.200, Z 556.000, A 0.000, B 90.000, C 0.000, E1 0.000, E2 0.0, E3 0.0, E4 0.0, E5 0.0, E6 0.0} C_DIS
LIN {E6POS: X 1196.000, Y -233.200, Z 556.000, A 0.000, B 90.000, C 0.000, E1 0.000, E2 0.0, E3 0.0, E4 0.0, E5 0.0, E6 0.0} C_DIS
LIN {E6POS: X 1196.000, Y -234.200, Z 556.000, A 0.000, B 90.000, C 0.000, E1 0.000, E2 0.0, E3 0.0, E4 0.0, E5 0.0, E6 0.0} C_DIS
LIN {E6POS: X 1196.000, Y -235.200, Z 556.000, A 0.000, B 90.000, C 0.000, E1 0.000, E2 0.0, E3 0.0, E4 0.0, E5 0.0, E6 0.0} C_DIS
LIN {E6POS: X 1196.000, Y -236.200, Z 556.000, A 0.000, B 90.000, C 0.000, E1 0.000, E2 0.0, E3 0.0, E4 0.0, E5 0.0, E6 0.0} C_DIS
LIN {E6POS: X 1196.000, Y -237.200, Z 556.000, A 0.000, B 90.000, C 0.000, E1 0.000, E2 0.0, E3 0.0, E4 0.0, E5 0.0, E6 0.0} C_DIS
LIN {E6POS: X 1196.000, Y -237.200, Z 557.000, A 0.000, B 90.000, C 0.000, E1 0.000, E2 0.0, E3 0.0, E4 0.0, E5 0.0, E6 0.0} C_DIS
LIN {E6POS: X 1197.000, Y -237.200, Z 557.000, A 0.000, B 90.000, C 0.000, E1 0.000, E2 0.0, E3 0.0, E4 0.0, E5 0.0, E6 0.0} C_DIS
LIN {E6POS: X 1198.000, Y -237.200, Z 557.000, A 0.000, B 90.000, C 0.000, E1 0.000, E2 0.0, E3 0.0, E4 0.0, E5 0.0, E6 0.0} C_DIS
LIN {E6POS: X 1199.000, Y -237.200, Z 557.000, A 0.000, B 90.000, C 0.000, E1 0.000, E2 0.0, E3 0.0, E4 0.0, E5 0.0, E6 0.0} C_DIS
LIN {E6POS: X 1200.000, Y -237.200, Z 557.000, A 0.000, B 90.000, C 0.000, E1 0.000, E2 0.0, E3 0.0, E4 0.0, E5 0.0, E6 0.0} C_DIS
LIN {E6POS: X 1201.000, Y -237.200, Z 557.000, A 0.000, B 90.000, C 0.000, E1 0.000, E2 0.0, E3 0.0, E4 0.0, E5 0.0, E6 0.0} C_DIS
LIN {E6POS: X 1201.000, Y -237.200, Z 557.000, A 0.000, B 90.000, C 0.000, E1 0.000, E2 0.0, E3 0.0, E4 0.0, E5 0.0, E6 0.0} C_DIS
LIN {E6POS: X 1201.000, Y -236.200, Z 557.000, A 0.000, B 90.000, C 0.000, E1 0.000, E2 0.0, E3 0.0, E4 0.0, E5 0.0, E6 0.0} C_DIS
LIN {E6POS: X 1201.000, Y -235.200, Z 557.000, A 0.000, B 90.000, C 0.000, E1 0.000, E2 0.0, E3 0.0, E4 0.0, E5 0.0, E6 0.0} C_DIS
LIN {E6POS: X 1201.000, Y -234.200, Z 557.000, A 0.000, B 90.000, C 0.000, E1 0.000, E2 0.0, E3 0.0, E4 0.0, E5 0.0, E6 0.0} C_DIS
LIN {E6POS: X 1201.000, Y -233.200, Z 557.000, A 0.000, B 90.000, C 0.000, E1 0.000, E2 0.0, E3 0.0, E4 0.0, E5 0.0, E6 0.0} C_DIS
LIN {E6POS: X 1201.000, Y -232.200, Z 557.000, A 0.000, B 90.000, C 0.000, E1 0.000, E2 0.0, E3 0.0, E4 0.0, E5 0.0, E6 0.0} C_DIS
LIN {E6POS: X 1201.000, Y -231.200, Z 557.000, A 0.000, B 90.000, C 0.000, E1 0.000, E2 0.0, E3 0.0, E4 0.0, E5 0.0, E6 0.0} C_DIS
LIN {E6POS: X 1201.000, Y -230.200, Z 557.000, A 0.000, B 90.000, C 0.000, E1 0.000, E2 0.0, E3 0.0, E4 0.0, E5 0.0, E6 0.0} C_DIS
LIN {E6POS: X 1201.000, Y -229.200, Z 557.000, A 0.000, B 90.000, C 0.000, E1 0.000, E2 0.0, E3 0.0, E4 0.0, E5 0.0, E6 0.0} C_DIS
LIN {E6POS: X 1201.000, Y -228.200, Z 557.000, A 0.000, B 90.000, C 0.000, E1 0.000, E2 0.0, E3 0.0, E4 0.0, E5 0.0, E6 0.0} C_DIS
LIN {E6POS: X 1201.000, Y -227.200, Z 557.000, A 0.000, B 90.000, C 0.000, E1 0.000, E2 0.0, E3 0.0, E4 0.0, E5 0.0, E6 0.0} C_DIS
LIN {E6POS: X 1201.000, Y -226.200, Z 557.000, A 0.000, B 90.000, C 0.000, E1 0.000, E2 0.0, E3 0.0, E4 0.0, E5 0.0, E6 0.0} C_DIS
LIN {E6POS: X 1201.000, Y -225.200, Z 557.000, A 0.000, B 90.000, C 0.000, E1 0.000, E2 0.0, E3 0.0, E4 0.0, E5 0.0, E6 0.0} C_DIS
LIN {E6POS: X 1201.000, Y -224.200, Z 557.000, A 0.000, B 90.000, C 0.000, E1 0.000, E2 0.0, E3 0.0, E4 0.0, E5 0.0, E6 0.0} C_DIS
LIN {E6POS: X 1201.000, Y -223.200, Z 557.000, A 0.000, B 90.000, C 0.000, E1 0.000, E2 0.0, E3 0.0, E4 0.0, E5 0.0, E6 0.0} C_DIS
LIN {E6POS: X 1201.000, Y -222.200, Z 557.000, A 0.000, B 90.000, C 0.000, E1 0.000, E2 0.0, E3 0.0, E4 0.0, E5 0.0, E6 0.0} C_DIS
LIN {E6POS: X 1201.000, Y -221.200, Z 557.000, A 0.000, B 90.000, C 0.000, E1 0.000, E2 0.0, E3 0.0, E4 0.0, E5 0.0, E6 0.0} C_DIS
LIN {E6POS: X 1201.000, Y -220.200, Z 557.000, A 0.000, B 90.000, C 0.000, E1 0.000, E2 0.0, E3 0.0, E4 0.0, E5 0.0, E6 0.0} C_DIS
LIN {E6POS: X 1201.000, Y -219.200, Z 557.000, A 0.000, B 90.000, C 0.000, E1 0.000, E2 0.0, E3 0.0, E4 0.0, E5 0.0, E6 0.0} C_DIS
LIN {E6POS: X 1201.000, Y -218.200, Z 557.000, A 0.000, B 90.000, C 0.000, E1 0.000, E2 0.0, E3 0.0, E4 0.0, E5 0.0, E6 0.0} C_DIS
LIN {E6POS: X 1201.000, Y -217.200, Z 557.000, A 0.000, B 90.000, C 0.000, E1 0.000, E2 0.0, E3 0.0, E4 0.0, E5 0.0, E6 0.0} C_DIS
LIN {E6POS: X 1201.000, Y -216.200, Z 557.000, A 0.000, B 90.000, C 0.000, E1 0.000, E2 0.0, E3 0.0, E4 0.0, E5 0.0, E6 0.0} C_DIS
LIN {E6POS: X 1201.000, Y -215.200, Z 557.000, A 0.000, B 90.000, C 0.000, E1 0.000, E2 0.0, E3 0.0, E4 0.0, E5 0.0, E6 0.0} C_DIS
LIN {E6POS: X 1201.000, Y -214.200, Z 557.000, A 0.000, B 90.000, C 0.000, E1 0.000, E2 0.0, E3 0.0, E4 0.0, E5 0.0, E6 0.0} C_DIS
LIN {E6POS: X 1201.000, Y -213.200, Z 557.000, A 0.000, B 90.000, C 0.000, E1 0.000, E2 0.0, E3 0.0, E4 0.0, E5 0.0, E6 0.0} C_DIS
LIN {E6POS: X 1201.000, Y -212.200, Z 557.000, A 0.000, B 90.000, C 0.000, E1 0.000, E2 0.0, E3 0.0, E4 0.0, E5 0.0, E6 0.0} C_DIS
LIN {E6POS: X 1201.000, Y -211.200, Z 557.000, A 0.000, B 90.000, C 0.000, E1 0.000, E2 0.0, E3 0.0, E4 0.0, E5 0.0, E6 0.0} C_DIS
LIN {E6POS: X 1201.000, Y -210.200, Z 557.000, A 0.000, B 90.000, C 0.000, E1 0.000, E2 0.0, E3 0.0, E4 0.0, E5 0.0, E6 0.0} C_DIS
LIN {E6POS: X 1201.000, Y -209.200, Z 557.000, A 0.000, B 90.000, C 0.000, E1 0.000, E2 0.0, E3 0.0, E4 0.0, E5 0.0, E6 0.0} C_DIS
LIN {E6POS: X 1201.000, Y -208.200, Z 557.000, A 0.000, B 90.000, C 0.000, E1 0.000, E2 0.0, E3 0.0, E4 0.0, E5 0.0, E6 0.0} C_DIS
LIN {E6POS: X 1201.000, Y -207.200, Z 557.000, A 0.000, B 90.000, C 0.000, E1 0.000, E2 0.0, E3 0.0, E4 0.0, E5 0.0, E6 0.0} C_DIS
LIN {E6POS: X 1201.000, Y -206.200, Z 557.000, A 0.000, B 90.000, C 0.000, E1 0.000, E2 0.0, E3 0.0, E4 0.0, E5 0.0, E6 0.0} C_DIS
LIN {E6POS: X 1201.000, Y -205.200, Z 557.000, A 0.000, B 90.000, C 0.000, E1 0.000, E2 0.0, E3 0.0, E4 0.0, E5 0.0, E6 0.0} C_DIS
LIN {E6POS: X 1201.000, Y -204.200, Z 557.000, A 0.000, B 90.000, C 0.000, E1 0.000, E2 0.0, E3 0.0, E4 0.0, E5 0.0, E6 0.0} C_DIS
LIN {E6POS: X 1201.000, Y -203.200, Z 557.000, A 0.000, B 90.000, C 0.000, E1 0.000, E2 0.0, E3 0.0, E4 0.0, E5 0.0, E6 0.0} C_DIS
LIN {E6POS: X 1201.000, Y -202.200, Z 557.000, A 0.000, B 90.000, C 0.000, E1 0.000, E2 0.0, E3 0.0, E4 0.0, E5 0.0, E6 0.0} C_DIS
LIN {E6POS: X 1201.000, Y -201.200, Z 557.000, A 0.000, B 90.000, C 0.000, E1 0.000, E2 0.0, E3 0.0, E4 0.0, E5 0.0, E6 0.0} C_DIS
LIN {E6POS: X 1201.000, Y -200.200, Z 557.000, A 0.000, B 90.000, C 0.000, E1 0.000, E2 0.0, E3 0.0, E4 0.0, E5 0.0, E6 0.0} C_DIS
LIN {E6POS: X 1201.000, Y -199.200, Z 557.000, A 0.000, B 90.000, C 0.000, E1 0.000, E2 0.0, E3 0.0, E4 0.0, E5 0.0, E6 0.0} C_DIS
LIN {E6POS: X 1201.000, Y -198.200, Z 557.000, A 0.000, B 90.000, C 0.000, E1 0.000, E2 0.0, E3 0.0, E4 0.0, E5 0.0, E6 0.0} C_DIS
LIN {E6POS: X 1201.000, Y -197.200, Z 557.000, A 0.000, B 90.000, C 0.000, E1 0.000, E2 0.0, E3 0.0, E4 0.0, E5 0.0, E6 0.0} C_DIS
LIN {E6POS: X 1201.000, Y -196.200, Z 557.000, A 0.000, B 90.000, C 0.000, E1 0.000, E2 0.0, E3 0.0, E4 0.0, E5 0.0, E6 0.0} C_DIS
LIN {E6POS: X 1201.000, Y -195.200, Z 557.000, A 0.000, B 90.000, C 0.000, E1 0.000, E2 0.0, E3 0.0, E4 0.0, E5 0.0, E6 0.0} C_DIS
LIN {E6POS: X 1201.000, Y -194.200, Z 557.000, A 0.000, B 90.000, C 0.000, E1 0.000, E2 0.0, E3 0.0, E4 0.0, E5 0.0, E6 0.0} C_DIS
LIN {E6POS: X 1201.000, Y -193.200, Z 557.000, A 0.000, B 90.000, C 0.000, E1 0.000, E2 0.0, E3 0.0, E4 0.0, E5 0.0, E6 0.0} C_DIS
LIN {E6POS: X 1201.000, Y -192.200, Z 557.000, A 0.000, B 90.000, C 0.000, E1 0.000, E2 0.0, E3 0.0, E4 0.0, E5 0.0, E6 0.0} C_DIS
LIN {E6POS: X 1201.000, Y -191.200, Z 557.000, A 0.000, B 90.000, C 0.000, E1 0.000, E2 0.0, E3 0.0, E4 0.0, E5 0.0, E6 0.0} C_DIS
LIN {E6POS: X 1201.000, Y -190.200, Z 557.000, A 0.000, B 90.000, C 0.000, E1 0.000, E2 0.0, E3 0.0, E4 0.0, E5 0.0, E6 0.0} C_DIS
LIN {E6POS: X 1201.000, Y -189.200, Z 557.000, A 0.000, B 90.000, C 0.000, E1 0.000, E2 0.0, E3 0.0, E4 0.0, E5 0.0, E6 0.0} C_DIS
LIN {E6POS: X 1201.000, Y -188.200, Z 557.000, A 0.000, B 90.000, C 0.000, E1 0.000, E2 0.0, E3 0.0, E4 0.0, E5 0.0, E6 0.0} C_DIS
LIN {E6POS: X 1201.000, Y -187.200, Z 557.000, A 0.000, B 90.000, C 0.000, E1 0.000, E2 0.0, E3 0.0, E4 0.0, E5 0.0, E6 0.0} C_DIS
LIN {E6POS: X 1201.000, Y -187.200, Z 557.000, A 0.000, B 90.000, C 0.000, E1 0.000, E2 0.0, E3 0.0, E4 0.0, E5 0.0, E6 0.0} C_DIS
LIN {E6POS: X 1200.000, Y -187.200, Z 557.000, A 0.000, B 90.000, C 0.000, E1 0.000, E2 0.0, E3 0.0, E4 0.0, E5 0.0, E6 0.0} C_DIS
LIN {E6POS: X 1199.000, Y -187.200, Z 557.000, A 0.000, B 90.000, C 0.000, E1 0.000, E2 0.0, E3 0.0, E4 0.0, E5 0.0, E6 0.0} C_DIS
LIN {E6POS: X 1198.000, Y -187.200, Z 557.000, A 0.000, B 90.000, C 0.000, E1 0.000, E2 0.0, E3 0.0, E4 0.0, E5 0.0, E6 0.0} C_DIS
LIN {E6POS: X 1197.000, Y -187.200, Z 557.000, A 0.000, B 90.000, C 0.000, E1 0.000, E2 0.0, E3 0.0, E4 0.0, E5 0.0, E6 0.0} C_DIS
LIN {E6POS: X 1196.000, Y -187.200, Z 557.000, A 0.000, B 90.000, C 0.000, E1 0.000, E2 0.0, E3 0.0, E4 0.0, E5 0.0, E6 0.0} C_DIS
LIN {E6POS: X 1196.000, Y -187.200, Z 557.000, A 0.000, B 90.000, C 0.000, E1 0.000, E2 0.0, E3 0.0, E4 0.0, E5 0.0, E6 0.0} C_DIS
LIN {E6POS: X 1196.000, Y -188.200, Z 557.000, A 0.000, B 90.000, C 0.000, E1 0.000, E2 0.0, E3 0.0, E4 0.0, E5 0.0, E6 0.0} C_DIS
LIN {E6POS: X 1196.000, Y -189.200, Z 557.000, A 0.000, B 90.000, C 0.000, E1 0.000, E2 0.0, E3 0.0, E4 0.0, E5 0.0, E6 0.0} C_DIS
LIN {E6POS: X 1196.000, Y -190.200, Z 557.000, A 0.000, B 90.000, C 0.000, E1 0.000, E2 0.0, E3 0.0, E4 0.0, E5 0.0, E6 0.0} C_DIS
LIN {E6POS: X 1196.000, Y -191.200, Z 557.000, A 0.000, B 90.000, C 0.000, E1 0.000, E2 0.0, E3 0.0, E4 0.0, E5 0.0, E6 0.0} C_DIS
LIN {E6POS: X 1196.000, Y -192.200, Z 557.000, A 0.000, B 90.000, C 0.000, E1 0.000, E2 0.0, E3 0.0, E4 0.0, E5 0.0, E6 0.0} C_DIS
LIN {E6POS: X 1196.000, Y -193.200, Z 557.000, A 0.000, B 90.000, C 0.000, E1 0.000, E2 0.0, E3 0.0, E4 0.0, E5 0.0, E6 0.0} C_DIS
LIN {E6POS: X 1196.000, Y -194.200, Z 557.000, A 0.000, B 90.000, C 0.000, E1 0.000, E2 0.0, E3 0.0, E4 0.0, E5 0.0, E6 0.0} C_DIS
LIN {E6POS: X 1196.000, Y -195.200, Z 557.000, A 0.000, B 90.000, C 0.000, E1 0.000, E2 0.0, E3 0.0, E4 0.0, E5 0.0, E6 0.0} C_DIS
LIN {E6POS: X 1196.000, Y -196.200, Z 557.000, A 0.000, B 90.000, C 0.000, E1 0.000, E2 0.0, E3 0.0, E4 0.0, E5 0.0, E6 0.0} C_DIS
LIN {E6POS: X 1196.000, Y -197.200, Z 557.000, A 0.000, B 90.000, C 0.000, E1 0.000, E2 0.0, E3 0.0, E4 0.0, E5 0.0, E6 0.0} C_DIS
LIN {E6POS: X 1196.000, Y -198.200, Z 557.000, A 0.000, B 90.000, C 0.000, E1 0.000, E2 0.0, E3 0.0, E4 0.0, E5 0.0, E6 0.0} C_DIS
LIN {E6POS: X 1196.000, Y -199.200, Z 557.000, A 0.000, B 90.000, C 0.000, E1 0.000, E2 0.0, E3 0.0, E4 0.0, E5 0.0, E6 0.0} C_DIS
LIN {E6POS: X 1196.000, Y -200.200, Z 557.000, A 0.000, B 90.000, C 0.000, E1 0.000, E2 0.0, E3 0.0, E4 0.0, E5 0.0, E6 0.0} C_DIS
LIN {E6POS: X 1196.000, Y -201.200, Z 557.000, A 0.000, B 90.000, C 0.000, E1 0.000, E2 0.0, E3 0.0, E4 0.0, E5 0.0, E6 0.0} C_DIS
LIN {E6POS: X 1196.000, Y -202.200, Z 557.000, A 0.000, B 90.000, C 0.000, E1 0.000, E2 0.0, E3 0.0, E4 0.0, E5 0.0, E6 0.0} C_DIS
LIN {E6POS: X 1196.000, Y -203.200, Z 557.000, A 0.000, B 90.000, C 0.000, E1 0.000, E2 0.0, E3 0.0, E4 0.0, E5 0.0, E6 0.0} C_DIS
LIN {E6POS: X 1196.000, Y -204.200, Z 557.000, A 0.000, B 90.000, C 0.000, E1 0.000, E2 0.0, E3 0.0, E4 0.0, E5 0.0, E6 0.0} C_DIS
LIN {E6POS: X 1196.000, Y -205.200, Z 557.000, A 0.000, B 90.000, C 0.000, E1 0.000, E2 0.0, E3 0.0, E4 0.0, E5 0.0, E6 0.0} C_DIS
LIN {E6POS: X 1196.000, Y -206.200, Z 557.000, A 0.000, B 90.000, C 0.000, E1 0.000, E2 0.0, E3 0.0, E4 0.0, E5 0.0, E6 0.0} C_DIS
LIN {E6POS: X 1196.000, Y -207.200, Z 557.000, A 0.000, B 90.000, C 0.000, E1 0.000, E2 0.0, E3 0.0, E4 0.0, E5 0.0, E6 0.0} C_DIS
LIN {E6POS: X 1196.000, Y -208.200, Z 557.000, A 0.000, B 90.000, C 0.000, E1 0.000, E2 0.0, E3 0.0, E4 0.0, E5 0.0, E6 0.0} C_DIS
LIN {E6POS: X 1196.000, Y -209.200, Z 557.000, A 0.000, B 90.000, C 0.000, E1 0.000, E2 0.0, E3 0.0, E4 0.0, E5 0.0, E6 0.0} C_DIS
LIN {E6POS: X 1196.000, Y -210.200, Z 557.000, A 0.000, B 90.000, C 0.000, E1 0.000, E2 0.0, E3 0.0, E4 0.0, E5 0.0, E6 0.0} C_DIS
LIN {E6POS: X 1196.000, Y -211.200, Z 557.000, A 0.000, B 90.000, C 0.000, E1 0.000, E2 0.0, E3 0.0, E4 0.0, E5 0.0, E6 0.0} C_DIS
LIN {E6POS: X 1196.000, Y -212.200, Z 557.000, A 0.000, B 90.000, C 0.000, E1 0.000, E2 0.0, E3 0.0, E4 0.0, E5 0.0, E6 0.0} C_DIS
LIN {E6POS: X 1196.000, Y -213.200, Z 557.000, A 0.000, B 90.000, C 0.000, E1 0.000, E2 0.0, E3 0.0, E4 0.0, E5 0.0, E6 0.0} C_DIS
LIN {E6POS: X 1196.000, Y -214.200, Z 557.000, A 0.000, B 90.000, C 0.000, E1 0.000, E2 0.0, E3 0.0, E4 0.0, E5 0.0, E6 0.0} C_DIS
LIN {E6POS: X 1196.000, Y -215.200, Z 557.000, A 0.000, B 90.000, C 0.000, E1 0.000, E2 0.0, E3 0.0, E4 0.0, E5 0.0, E6 0.0} C_DIS
LIN {E6POS: X 1196.000, Y -216.200, Z 557.000, A 0.000, B 90.000, C 0.000, E1 0.000, E2 0.0, E3 0.0, E4 0.0, E5 0.0, E6 0.0} C_DIS
LIN {E6POS: X 1196.000, Y -217.200, Z 557.000, A 0.000, B 90.000, C 0.000, E1 0.000, E2 0.0, E3 0.0, E4 0.0, E5 0.0, E6 0.0} C_DIS
LIN {E6POS: X 1196.000, Y -218.200, Z 557.000, A 0.000, B 90.000, C 0.000, E1 0.000, E2 0.0, E3 0.0, E4 0.0, E5 0.0, E6 0.0} C_DIS
LIN {E6POS: X 1196.000, Y -219.200, Z 557.000, A 0.000, B 90.000, C 0.000, E1 0.000, E2 0.0, E3 0.0, E4 0.0, E5 0.0, E6 0.0} C_DIS
LIN {E6POS: X 1196.000, Y -220.200, Z 557.000, A 0.000, B 90.000, C 0.000, E1 0.000, E2 0.0, E3 0.0, E4 0.0, E5 0.0, E6 0.0} C_DIS
LIN {E6POS: X 1196.000, Y -221.200, Z 557.000, A 0.000, B 90.000, C 0.000, E1 0.000, E2 0.0, E3 0.0, E4 0.0, E5 0.0, E6 0.0} C_DIS
LIN {E6POS: X 1196.000, Y -222.200, Z 557.000, A 0.000, B 90.000, C 0.000, E1 0.000, E2 0.0, E3 0.0, E4 0.0, E5 0.0, E6 0.0} C_DIS
LIN {E6POS: X 1196.000, Y -223.200, Z 557.000, A 0.000, B 90.000, C 0.000, E1 0.000, E2 0.0, E3 0.0, E4 0.0, E5 0.0, E6 0.0} C_DIS
LIN {E6POS: X 1196.000, Y -224.200, Z 557.000, A 0.000, B 90.000, C 0.000, E1 0.000, E2 0.0, E3 0.0, E4 0.0, E5 0.0, E6 0.0} C_DIS
LIN {E6POS: X 1196.000, Y -225.200, Z 557.000, A 0.000, B 90.000, C 0.000, E1 0.000, E2 0.0, E3 0.0, E4 0.0, E5 0.0, E6 0.0} C_DIS
LIN {E6POS: X 1196.000, Y -226.200, Z 557.000, A 0.000, B 90.000, C 0.000, E1 0.000, E2 0.0, E3 0.0, E4 0.0, E5 0.0, E6 0.0} C_DIS
LIN {E6POS: X 1196.000, Y -227.200, Z 557.000, A 0.000, B 90.000, C 0.000, E1 0.000, E2 0.0, E3 0.0, E4 0.0, E5 0.0, E6 0.0} C_DIS
LIN {E6POS: X 1196.000, Y -228.200, Z 557.000, A 0.000, B 90.000, C 0.000, E1 0.000, E2 0.0, E3 0.0, E4 0.0, E5 0.0, E6 0.0} C_DIS
LIN {E6POS: X 1196.000, Y -229.200, Z 557.000, A 0.000, B 90.000, C 0.000, E1 0.000, E2 0.0, E3 0.0, E4 0.0, E5 0.0, E6 0.0} C_DIS
LIN {E6POS: X 1196.000, Y -230.200, Z 557.000, A 0.000, B 90.000, C 0.000, E1 0.000, E2 0.0, E3 0.0, E4 0.0, E5 0.0, E6 0.0} C_DIS
LIN {E6POS: X 1196.000, Y -231.200, Z 557.000, A 0.000, B 90.000, C 0.000, E1 0.000, E2 0.0, E3 0.0, E4 0.0, E5 0.0, E6 0.0} C_DIS
LIN {E6POS: X 1196.000, Y -232.200, Z 557.000, A 0.000, B 90.000, C 0.000, E1 0.000, E2 0.0, E3 0.0, E4 0.0, E5 0.0, E6 0.0} C_DIS
LIN {E6POS: X 1196.000, Y -233.200, Z 557.000, A 0.000, B 90.000, C 0.000, E1 0.000, E2 0.0, E3 0.0, E4 0.0, E5 0.0, E6 0.0} C_DIS
LIN {E6POS: X 1196.000, Y -234.200, Z 557.000, A 0.000, B 90.000, C 0.000, E1 0.000, E2 0.0, E3 0.0, E4 0.0, E5 0.0, E6 0.0} C_DIS
LIN {E6POS: X 1196.000, Y -235.200, Z 557.000, A 0.000, B 90.000, C 0.000, E1 0.000, E2 0.0, E3 0.0, E4 0.0, E5 0.0, E6 0.0} C_DIS
LIN {E6POS: X 1196.000, Y -236.200, Z 557.000, A 0.000, B 90.000, C 0.000, E1 0.000, E2 0.0, E3 0.0, E4 0.0, E5 0.0, E6 0.0} C_DIS
LIN {E6POS: X 1196.000, Y -237.200, Z 557.000, A 0.000, B 90.000, C 0.000, E1 0.000, E2 0.0, E3 0.0, E4 0.0, E5 0.0, E6 0.0} C_DIS
LIN {E6POS: X 1196.000, Y -237.200, Z 558.000, A 0.000, B 90.000, C 0.000, E1 0.000, E2 0.0, E3 0.0, E4 0.0, E5 0.0, E6 0.0} C_DIS
LIN {E6POS: X 1197.000, Y -237.200, Z 558.000, A 0.000, B 90.000, C 0.000, E1 0.000, E2 0.0, E3 0.0, E4 0.0, E5 0.0, E6 0.0} C_DIS
LIN {E6POS: X 1198.000, Y -237.200, Z 558.000, A 0.000, B 90.000, C 0.000, E1 0.000, E2 0.0, E3 0.0, E4 0.0, E5 0.0, E6 0.0} C_DIS
LIN {E6POS: X 1199.000, Y -237.200, Z 558.000, A 0.000, B 90.000, C 0.000, E1 0.000, E2 0.0, E3 0.0, E4 0.0, E5 0.0, E6 0.0} C_DIS
LIN {E6POS: X 1200.000, Y -237.200, Z 558.000, A 0.000, B 90.000, C 0.000, E1 0.000, E2 0.0, E3 0.0, E4 0.0, E5 0.0, E6 0.0} C_DIS
LIN {E6POS: X 1201.000, Y -237.200, Z 558.000, A 0.000, B 90.000, C 0.000, E1 0.000, E2 0.0, E3 0.0, E4 0.0, E5 0.0, E6 0.0} C_DIS
LIN {E6POS: X 1201.000, Y -237.200, Z 558.000, A 0.000, B 90.000, C 0.000, E1 0.000, E2 0.0, E3 0.0, E4 0.0, E5 0.0, E6 0.0} C_DIS
LIN {E6POS: X 1201.000, Y -236.200, Z 558.000, A 0.000, B 90.000, C 0.000, E1 0.000, E2 0.0, E3 0.0, E4 0.0, E5 0.0, E6 0.0} C_DIS
LIN {E6POS: X 1201.000, Y -235.200, Z 558.000, A 0.000, B 90.000, C 0.000, E1 0.000, E2 0.0, E3 0.0, E4 0.0, E5 0.0, E6 0.0} C_DIS
LIN {E6POS: X 1201.000, Y -234.200, Z 558.000, A 0.000, B 90.000, C 0.000, E1 0.000, E2 0.0, E3 0.0, E4 0.0, E5 0.0, E6 0.0} C_DIS
LIN {E6POS: X 1201.000, Y -233.200, Z 558.000, A 0.000, B 90.000, C 0.000, E1 0.000, E2 0.0, E3 0.0, E4 0.0, E5 0.0, E6 0.0} C_DIS
LIN {E6POS: X 1201.000, Y -232.200, Z 558.000, A 0.000, B 90.000, C 0.000, E1 0.000, E2 0.0, E3 0.0, E4 0.0, E5 0.0, E6 0.0} C_DIS
LIN {E6POS: X 1201.000, Y -231.200, Z 558.000, A 0.000, B 90.000, C 0.000, E1 0.000, E2 0.0, E3 0.0, E4 0.0, E5 0.0, E6 0.0} C_DIS
LIN {E6POS: X 1201.000, Y -230.200, Z 558.000, A 0.000, B 90.000, C 0.000, E1 0.000, E2 0.0, E3 0.0, E4 0.0, E5 0.0, E6 0.0} C_DIS
LIN {E6POS: X 1201.000, Y -229.200, Z 558.000, A 0.000, B 90.000, C 0.000, E1 0.000, E2 0.0, E3 0.0, E4 0.0, E5 0.0, E6 0.0} C_DIS
LIN {E6POS: X 1201.000, Y -228.200, Z 558.000, A 0.000, B 90.000, C 0.000, E1 0.000, E2 0.0, E3 0.0, E4 0.0, E5 0.0, E6 0.0} C_DIS
LIN {E6POS: X 1201.000, Y -227.200, Z 558.000, A 0.000, B 90.000, C 0.000, E1 0.000, E2 0.0, E3 0.0, E4 0.0, E5 0.0, E6 0.0} C_DIS
LIN {E6POS: X 1201.000, Y -226.200, Z 558.000, A 0.000, B 90.000, C 0.000, E1 0.000, E2 0.0, E3 0.0, E4 0.0, E5 0.0, E6 0.0} C_DIS
LIN {E6POS: X 1201.000, Y -225.200, Z 558.000, A 0.000, B 90.000, C 0.000, E1 0.000, E2 0.0, E3 0.0, E4 0.0, E5 0.0, E6 0.0} C_DIS
LIN {E6POS: X 1201.000, Y -224.200, Z 558.000, A 0.000, B 90.000, C 0.000, E1 0.000, E2 0.0, E3 0.0, E4 0.0, E5 0.0, E6 0.0} C_DIS
LIN {E6POS: X 1201.000, Y -223.200, Z 558.000, A 0.000, B 90.000, C 0.000, E1 0.000, E2 0.0, E3 0.0, E4 0.0, E5 0.0, E6 0.0} C_DIS
LIN {E6POS: X 1201.000, Y -222.200, Z 558.000, A 0.000, B 90.000, C 0.000, E1 0.000, E2 0.0, E3 0.0, E4 0.0, E5 0.0, E6 0.0} C_DIS
LIN {E6POS: X 1201.000, Y -221.200, Z 558.000, A 0.000, B 90.000, C 0.000, E1 0.000, E2 0.0, E3 0.0, E4 0.0, E5 0.0, E6 0.0} C_DIS
LIN {E6POS: X 1201.000, Y -220.200, Z 558.000, A 0.000, B 90.000, C 0.000, E1 0.000, E2 0.0, E3 0.0, E4 0.0, E5 0.0, E6 0.0} C_DIS
LIN {E6POS: X 1201.000, Y -219.200, Z 558.000, A 0.000, B 90.000, C 0.000, E1 0.000, E2 0.0, E3 0.0, E4 0.0, E5 0.0, E6 0.0} C_DIS
LIN {E6POS: X 1201.000, Y -218.200, Z 558.000, A 0.000, B 90.000, C 0.000, E1 0.000, E2 0.0, E3 0.0, E4 0.0, E5 0.0, E6 0.0} C_DIS
LIN {E6POS: X 1201.000, Y -217.200, Z 558.000, A 0.000, B 90.000, C 0.000, E1 0.000, E2 0.0, E3 0.0, E4 0.0, E5 0.0, E6 0.0} C_DIS
LIN {E6POS: X 1201.000, Y -216.200, Z 558.000, A 0.000, B 90.000, C 0.000, E1 0.000, E2 0.0, E3 0.0, E4 0.0, E5 0.0, E6 0.0} C_DIS
LIN {E6POS: X 1201.000, Y -215.200, Z 558.000, A 0.000, B 90.000, C 0.000, E1 0.000, E2 0.0, E3 0.0, E4 0.0, E5 0.0, E6 0.0} C_DIS
LIN {E6POS: X 1201.000, Y -214.200, Z 558.000, A 0.000, B 90.000, C 0.000, E1 0.000, E2 0.0, E3 0.0, E4 0.0, E5 0.0, E6 0.0} C_DIS
LIN {E6POS: X 1201.000, Y -213.200, Z 558.000, A 0.000, B 90.000, C 0.000, E1 0.000, E2 0.0, E3 0.0, E4 0.0, E5 0.0, E6 0.0} C_DIS
LIN {E6POS: X 1201.000, Y -212.200, Z 558.000, A 0.000, B 90.000, C 0.000, E1 0.000, E2 0.0, E3 0.0, E4 0.0, E5 0.0, E6 0.0} C_DIS
LIN {E6POS: X 1201.000, Y -211.200, Z 558.000, A 0.000, B 90.000, C 0.000, E1 0.000, E2 0.0, E3 0.0, E4 0.0, E5 0.0, E6 0.0} C_DIS
LIN {E6POS: X 1201.000, Y -210.200, Z 558.000, A 0.000, B 90.000, C 0.000, E1 0.000, E2 0.0, E3 0.0, E4 0.0, E5 0.0, E6 0.0} C_DIS
LIN {E6POS: X 1201.000, Y -209.200, Z 558.000, A 0.000, B 90.000, C 0.000, E1 0.000, E2 0.0, E3 0.0, E4 0.0, E5 0.0, E6 0.0} C_DIS
LIN {E6POS: X 1201.000, Y -208.200, Z 558.000, A 0.000, B 90.000, C 0.000, E1 0.000, E2 0.0, E3 0.0, E4 0.0, E5 0.0, E6 0.0} C_DIS
LIN {E6POS: X 1201.000, Y -207.200, Z 558.000, A 0.000, B 90.000, C 0.000, E1 0.000, E2 0.0, E3 0.0, E4 0.0, E5 0.0, E6 0.0} C_DIS
LIN {E6POS: X 1201.000, Y -206.200, Z 558.000, A 0.000, B 90.000, C 0.000, E1 0.000, E2 0.0, E3 0.0, E4 0.0, E5 0.0, E6 0.0} C_DIS
LIN {E6POS: X 1201.000, Y -205.200, Z 558.000, A 0.000, B 90.000, C 0.000, E1 0.000, E2 0.0, E3 0.0, E4 0.0, E5 0.0, E6 0.0} C_DIS
LIN {E6POS: X 1201.000, Y -204.200, Z 558.000, A 0.000, B 90.000, C 0.000, E1 0.000, E2 0.0, E3 0.0, E4 0.0, E5 0.0, E6 0.0} C_DIS
LIN {E6POS: X 1201.000, Y -203.200, Z 558.000, A 0.000, B 90.000, C 0.000, E1 0.000, E2 0.0, E3 0.0, E4 0.0, E5 0.0, E6 0.0} C_DIS
LIN {E6POS: X 1201.000, Y -202.200, Z 558.000, A 0.000, B 90.000, C 0.000, E1 0.000, E2 0.0, E3 0.0, E4 0.0, E5 0.0, E6 0.0} C_DIS
LIN {E6POS: X 1201.000, Y -201.200, Z 558.000, A 0.000, B 90.000, C 0.000, E1 0.000, E2 0.0, E3 0.0, E4 0.0, E5 0.0, E6 0.0} C_DIS
LIN {E6POS: X 1201.000, Y -200.200, Z 558.000, A 0.000, B 90.000, C 0.000, E1 0.000, E2 0.0, E3 0.0, E4 0.0, E5 0.0, E6 0.0} C_DIS
LIN {E6POS: X 1201.000, Y -199.200, Z 558.000, A 0.000, B 90.000, C 0.000, E1 0.000, E2 0.0, E3 0.0, E4 0.0, E5 0.0, E6 0.0} C_DIS
LIN {E6POS: X 1201.000, Y -198.200, Z 558.000, A 0.000, B 90.000, C 0.000, E1 0.000, E2 0.0, E3 0.0, E4 0.0, E5 0.0, E6 0.0} C_DIS
LIN {E6POS: X 1201.000, Y -197.200, Z 558.000, A 0.000, B 90.000, C 0.000, E1 0.000, E2 0.0, E3 0.0, E4 0.0, E5 0.0, E6 0.0} C_DIS
LIN {E6POS: X 1201.000, Y -196.200, Z 558.000, A 0.000, B 90.000, C 0.000, E1 0.000, E2 0.0, E3 0.0, E4 0.0, E5 0.0, E6 0.0} C_DIS
LIN {E6POS: X 1201.000, Y -195.200, Z 558.000, A 0.000, B 90.000, C 0.000, E1 0.000, E2 0.0, E3 0.0, E4 0.0, E5 0.0, E6 0.0} C_DIS
LIN {E6POS: X 1201.000, Y -194.200, Z 558.000, A 0.000, B 90.000, C 0.000, E1 0.000, E2 0.0, E3 0.0, E4 0.0, E5 0.0, E6 0.0} C_DIS
LIN {E6POS: X 1201.000, Y -193.200, Z 558.000, A 0.000, B 90.000, C 0.000, E1 0.000, E2 0.0, E3 0.0, E4 0.0, E5 0.0, E6 0.0} C_DIS
LIN {E6POS: X 1201.000, Y -192.200, Z 558.000, A 0.000, B 90.000, C 0.000, E1 0.000, E2 0.0, E3 0.0, E4 0.0, E5 0.0, E6 0.0} C_DIS
LIN {E6POS: X 1201.000, Y -191.200, Z 558.000, A 0.000, B 90.000, C 0.000, E1 0.000, E2 0.0, E3 0.0, E4 0.0, E5 0.0, E6 0.0} C_DIS
LIN {E6POS: X 1201.000, Y -190.200, Z 558.000, A 0.000, B 90.000, C 0.000, E1 0.000, E2 0.0, E3 0.0, E4 0.0, E5 0.0, E6 0.0} C_DIS
LIN {E6POS: X 1201.000, Y -189.200, Z 558.000, A 0.000, B 90.000, C 0.000, E1 0.000, E2 0.0, E3 0.0, E4 0.0, E5 0.0, E6 0.0} C_DIS
LIN {E6POS: X 1201.000, Y -188.200, Z 558.000, A 0.000, B 90.000, C 0.000, E1 0.000, E2 0.0, E3 0.0, E4 0.0, E5 0.0, E6 0.0} C_DIS
LIN {E6POS: X 1201.000, Y -187.200, Z 558.000, A 0.000, B 90.000, C 0.000, E1 0.000, E2 0.0, E3 0.0, E4 0.0, E5 0.0, E6 0.0} C_DIS
LIN {E6POS: X 1201.000, Y -187.200, Z 558.000, A 0.000, B 90.000, C 0.000, E1 0.000, E2 0.0, E3 0.0, E4 0.0, E5 0.0, E6 0.0} C_DIS
LIN {E6POS: X 1200.000, Y -187.200, Z 558.000, A 0.000, B 90.000, C 0.000, E1 0.000, E2 0.0, E3 0.0, E4 0.0, E5 0.0, E6 0.0} C_DIS
LIN {E6POS: X 1199.000, Y -187.200, Z 558.000, A 0.000, B 90.000, C 0.000, E1 0.000, E2 0.0, E3 0.0, E4 0.0, E5 0.0, E6 0.0} C_DIS
LIN {E6POS: X 1198.000, Y -187.200, Z 558.000, A 0.000, B 90.000, C 0.000, E1 0.000, E2 0.0, E3 0.0, E4 0.0, E5 0.0, E6 0.0} C_DIS
LIN {E6POS: X 1197.000, Y -187.200, Z 558.000, A 0.000, B 90.000, C 0.000, E1 0.000, E2 0.0, E3 0.0, E4 0.0, E5 0.0, E6 0.0} C_DIS
LIN {E6POS: X 1196.000, Y -187.200, Z 558.000, A 0.000, B 90.000, C 0.000, E1 0.000, E2 0.0, E3 0.0, E4 0.0, E5 0.0, E6 0.0} C_DIS
LIN {E6POS: X 1196.000, Y -187.200, Z 558.000, A 0.000, B 90.000, C 0.000, E1 0.000, E2 0.0, E3 0.0, E4 0.0, E5 0.0, E6 0.0} C_DIS
LIN {E6POS: X 1196.000, Y -188.200, Z 558.000, A 0.000, B 90.000, C 0.000, E1 0.000, E2 0.0, E3 0.0, E4 0.0, E5 0.0, E6 0.0} C_DIS
LIN {E6POS: X 1196.000, Y -189.200, Z 558.000, A 0.000, B 90.000, C 0.000, E1 0.000, E2 0.0, E3 0.0, E4 0.0, E5 0.0, E6 0.0} C_DIS
LIN {E6POS: X 1196.000, Y -190.200, Z 558.000, A 0.000, B 90.000, C 0.000, E1 0.000, E2 0.0, E3 0.0, E4 0.0, E5 0.0, E6 0.0} C_DIS
LIN {E6POS: X 1196.000, Y -191.200, Z 558.000, A 0.000, B 90.000, C 0.000, E1 0.000, E2 0.0, E3 0.0, E4 0.0, E5 0.0, E6 0.0} C_DIS
LIN {E6POS: X 1196.000, Y -192.200, Z 558.000, A 0.000, B 90.000, C 0.000, E1 0.000, E2 0.0, E3 0.0, E4 0.0, E5 0.0, E6 0.0} C_DIS
LIN {E6POS: X 1196.000, Y -193.200, Z 558.000, A 0.000, B 90.000, C 0.000, E1 0.000, E2 0.0, E3 0.0, E4 0.0, E5 0.0, E6 0.0} C_DIS
LIN {E6POS: X 1196.000, Y -194.200, Z 558.000, A 0.000, B 90.000, C 0.000, E1 0.000, E2 0.0, E3 0.0, E4 0.0, E5 0.0, E6 0.0} C_DIS
LIN {E6POS: X 1196.000, Y -195.200, Z 558.000, A 0.000, B 90.000, C 0.000, E1 0.000, E2 0.0, E3 0.0, E4 0.0, E5 0.0, E6 0.0} C_DIS
LIN {E6POS: X 1196.000, Y -196.200, Z 558.000, A 0.000, B 90.000, C 0.000, E1 0.000, E2 0.0, E3 0.0, E4 0.0, E5 0.0, E6 0.0} C_DIS
LIN {E6POS: X 1196.000, Y -197.200, Z 558.000, A 0.000, B 90.000, C 0.000, E1 0.000, E2 0.0, E3 0.0, E4 0.0, E5 0.0, E6 0.0} C_DIS
LIN {E6POS: X 1196.000, Y -198.200, Z 558.000, A 0.000, B 90.000, C 0.000, E1 0.000, E2 0.0, E3 0.0, E4 0.0, E5 0.0, E6 0.0} C_DIS
LIN {E6POS: X 1196.000, Y -199.200, Z 558.000, A 0.000, B 90.000, C 0.000, E1 0.000, E2 0.0, E3 0.0, E4 0.0, E5 0.0, E6 0.0} C_DIS
LIN {E6POS: X 1196.000, Y -200.200, Z 558.000, A 0.000, B 90.000, C 0.000, E1 0.000, E2 0.0, E3 0.0, E4 0.0, E5 0.0, E6 0.0} C_DIS
LIN {E6POS: X 1196.000, Y -201.200, Z 558.000, A 0.000, B 90.000, C 0.000, E1 0.000, E2 0.0, E3 0.0, E4 0.0, E5 0.0, E6 0.0} C_DIS
LIN {E6POS: X 1196.000, Y -202.200, Z 558.000, A 0.000, B 90.000, C 0.000, E1 0.000, E2 0.0, E3 0.0, E4 0.0, E5 0.0, E6 0.0} C_DIS
LIN {E6POS: X 1196.000, Y -203.200, Z 558.000, A 0.000, B 90.000, C 0.000, E1 0.000, E2 0.0, E3 0.0, E4 0.0, E5 0.0, E6 0.0} C_DIS
LIN {E6POS: X 1196.000, Y -204.200, Z 558.000, A 0.000, B 90.000, C 0.000, E1 0.000, E2 0.0, E3 0.0, E4 0.0, E5 0.0, E6 0.0} C_DIS
LIN {E6POS: X 1196.000, Y -205.200, Z 558.000, A 0.000, B 90.000, C 0.000, E1 0.000, E2 0.0, E3 0.0, E4 0.0, E5 0.0, E6 0.0} C_DIS
LIN {E6POS: X 1196.000, Y -206.200, Z 558.000, A 0.000, B 90.000, C 0.000, E1 0.000, E2 0.0, E3 0.0, E4 0.0, E5 0.0, E6 0.0} C_DIS
LIN {E6POS: X 1196.000, Y -207.200, Z 558.000, A 0.000, B 90.000, C 0.000, E1 0.000, E2 0.0, E3 0.0, E4 0.0, E5 0.0, E6 0.0} C_DIS
LIN {E6POS: X 1196.000, Y -208.200, Z 558.000, A 0.000, B 90.000, C 0.000, E1 0.000, E2 0.0, E3 0.0, E4 0.0, E5 0.0, E6 0.0} C_DIS
LIN {E6POS: X 1196.000, Y -209.200, Z 558.000, A 0.000, B 90.000, C 0.000, E1 0.000, E2 0.0, E3 0.0, E4 0.0, E5 0.0, E6 0.0} C_DIS
LIN {E6POS: X 1196.000, Y -210.200, Z 558.000, A 0.000, B 90.000, C 0.000, E1 0.000, E2 0.0, E3 0.0, E4 0.0, E5 0.0, E6 0.0} C_DIS
LIN {E6POS: X 1196.000, Y -211.200, Z 558.000, A 0.000, B 90.000, C 0.000, E1 0.000, E2 0.0, E3 0.0, E4 0.0, E5 0.0, E6 0.0} C_DIS
LIN {E6POS: X 1196.000, Y -212.200, Z 558.000, A 0.000, B 90.000, C 0.000, E1 0.000, E2 0.0, E3 0.0, E4 0.0, E5 0.0, E6 0.0} C_DIS
LIN {E6POS: X 1196.000, Y -213.200, Z 558.000, A 0.000, B 90.000, C 0.000, E1 0.000, E2 0.0, E3 0.0, E4 0.0, E5 0.0, E6 0.0} C_DIS
LIN {E6POS: X 1196.000, Y -214.200, Z 558.000, A 0.000, B 90.000, C 0.000, E1 0.000, E2 0.0, E3 0.0, E4 0.0, E5 0.0, E6 0.0} C_DIS
LIN {E6POS: X 1196.000, Y -215.200, Z 558.000, A 0.000, B 90.000, C 0.000, E1 0.000, E2 0.0, E3 0.0, E4 0.0, E5 0.0, E6 0.0} C_DIS
LIN {E6POS: X 1196.000, Y -216.200, Z 558.000, A 0.000, B 90.000, C 0.000, E1 0.000, E2 0.0, E3 0.0, E4 0.0, E5 0.0, E6 0.0} C_DIS
LIN {E6POS: X 1196.000, Y -217.200, Z 558.000, A 0.000, B 90.000, C 0.000, E1 0.000, E2 0.0, E3 0.0, E4 0.0, E5 0.0, E6 0.0} C_DIS
LIN {E6POS: X 1196.000, Y -218.200, Z 558.000, A 0.000, B 90.000, C 0.000, E1 0.000, E2 0.0, E3 0.0, E4 0.0, E5 0.0, E6 0.0} C_DIS
LIN {E6POS: X 1196.000, Y -219.200, Z 558.000, A 0.000, B 90.000, C 0.000, E1 0.000, E2 0.0, E3 0.0, E4 0.0, E5 0.0, E6 0.0} C_DIS
LIN {E6POS: X 1196.000, Y -220.200, Z 558.000, A 0.000, B 90.000, C 0.000, E1 0.000, E2 0.0, E3 0.0, E4 0.0, E5 0.0, E6 0.0} C_DIS
LIN {E6POS: X 1196.000, Y -221.200, Z 558.000, A 0.000, B 90.000, C 0.000, E1 0.000, E2 0.0, E3 0.0, E4 0.0, E5 0.0, E6 0.0} C_DIS
LIN {E6POS: X 1196.000, Y -222.200, Z 558.000, A 0.000, B 90.000, C 0.000, E1 0.000, E2 0.0, E3 0.0, E4 0.0, E5 0.0, E6 0.0} C_DIS
LIN {E6POS: X 1196.000, Y -223.200, Z 558.000, A 0.000, B 90.000, C 0.000, E1 0.000, E2 0.0, E3 0.0, E4 0.0, E5 0.0, E6 0.0} C_DIS
LIN {E6POS: X 1196.000, Y -224.200, Z 558.000, A 0.000, B 90.000, C 0.000, E1 0.000, E2 0.0, E3 0.0, E4 0.0, E5 0.0, E6 0.0} C_DIS
LIN {E6POS: X 1196.000, Y -225.200, Z 558.000, A 0.000, B 90.000, C 0.000, E1 0.000, E2 0.0, E3 0.0, E4 0.0, E5 0.0, E6 0.0} C_DIS
LIN {E6POS: X 1196.000, Y -226.200, Z 558.000, A 0.000, B 90.000, C 0.000, E1 0.000, E2 0.0, E3 0.0, E4 0.0, E5 0.0, E6 0.0} C_DIS
LIN {E6POS: X 1196.000, Y -227.200, Z 558.000, A 0.000, B 90.000, C 0.000, E1 0.000, E2 0.0, E3 0.0, E4 0.0, E5 0.0, E6 0.0} C_DIS
LIN {E6POS: X 1196.000, Y -228.200, Z 558.000, A 0.000, B 90.000, C 0.000, E1 0.000, E2 0.0, E3 0.0, E4 0.0, E5 0.0, E6 0.0} C_DIS
LIN {E6POS: X 1196.000, Y -229.200, Z 558.000, A 0.000, B 90.000, C 0.000, E1 0.000, E2 0.0, E3 0.0, E4 0.0, E5 0.0, E6 0.0} C_DIS
LIN {E6POS: X 1196.000, Y -230.200, Z 558.000, A 0.000, B 90.000, C 0.000, E1 0.000, E2 0.0, E3 0.0, E4 0.0, E5 0.0, E6 0.0} C_DIS
LIN {E6POS: X 1196.000, Y -231.200, Z 558.000, A 0.000, B 90.000, C 0.000, E1 0.000, E2 0.0, E3 0.0, E4 0.0, E5 0.0, E6 0.0} C_DIS
LIN {E6POS: X 1196.000, Y -232.200, Z 558.000, A 0.000, B 90.000, C 0.000, E1 0.000, E2 0.0, E3 0.0, E4 0.0, E5 0.0, E6 0.0} C_DIS
LIN {E6POS: X 1196.000, Y -233.200, Z 558.000, A 0.000, B 90.000, C 0.000, E1 0.000, E2 0.0, E3 0.0, E4 0.0, E5 0.0, E6 0.0} C_DIS
LIN {E6POS: X 1196.000, Y -234.200, Z 558.000, A 0.000, B 90.000, C 0.000, E1 0.000, E2 0.0, E3 0.0, E4 0.0, E5 0.0, E6 0.0} C_DIS
LIN {E6POS: X 1196.000, Y -235.200, Z 558.000, A 0.000, B 90.000, C 0.000, E1 0.000, E2 0.0, E3 0.0, E4 0.0, E5 0.0, E6 0.0} C_DIS
LIN {E6POS: X 1196.000, Y -236.200, Z 558.000, A 0.000, B 90.000, C 0.000, E1 0.000, E2 0.0, E3 0.0, E4 0.0, E5 0.0, E6 0.0} C_DIS
LIN {E6POS: X 1196.000, Y -237.200, Z 558.000, A 0.000, B 90.000, C 0.000, E1 0.000, E2 0.0, E3 0.0, E4 0.0, E5 0.0, E6 0.0} C_DIS
LIN {E6POS: X 1196.000, Y -237.200, Z 559.000, A 0.000, B 90.000, C 0.000, E1 0.000, E2 0.0, E3 0.0, E4 0.0, E5 0.0, E6 0.0} C_DIS
LIN {E6POS: X 1197.000, Y -237.200, Z 559.000, A 0.000, B 90.000, C 0.000, E1 0.000, E2 0.0, E3 0.0, E4 0.0, E5 0.0, E6 0.0} C_DIS
LIN {E6POS: X 1198.000, Y -237.200, Z 559.000, A 0.000, B 90.000, C 0.000, E1 0.000, E2 0.0, E3 0.0, E4 0.0, E5 0.0, E6 0.0} C_DIS
LIN {E6POS: X 1199.000, Y -237.200, Z 559.000, A 0.000, B 90.000, C 0.000, E1 0.000, E2 0.0, E3 0.0, E4 0.0, E5 0.0, E6 0.0} C_DIS
LIN {E6POS: X 1200.000, Y -237.200, Z 559.000, A 0.000, B 90.000, C 0.000, E1 0.000, E2 0.0, E3 0.0, E4 0.0, E5 0.0, E6 0.0} C_DIS
LIN {E6POS: X 1201.000, Y -237.200, Z 559.000, A 0.000, B 90.000, C 0.000, E1 0.000, E2 0.0, E3 0.0, E4 0.0, E5 0.0, E6 0.0} C_DIS
LIN {E6POS: X 1201.000, Y -237.200, Z 559.000, A 0.000, B 90.000, C 0.000, E1 0.000, E2 0.0, E3 0.0, E4 0.0, E5 0.0, E6 0.0} C_DIS
LIN {E6POS: X 1201.000, Y -236.200, Z 559.000, A 0.000, B 90.000, C 0.000, E1 0.000, E2 0.0, E3 0.0, E4 0.0, E5 0.0, E6 0.0} C_DIS
LIN {E6POS: X 1201.000, Y -235.200, Z 559.000, A 0.000, B 90.000, C 0.000, E1 0.000, E2 0.0, E3 0.0, E4 0.0, E5 0.0, E6 0.0} C_DIS
LIN {E6POS: X 1201.000, Y -234.200, Z 559.000, A 0.000, B 90.000, C 0.000, E1 0.000, E2 0.0, E3 0.0, E4 0.0, E5 0.0, E6 0.0} C_DIS
LIN {E6POS: X 1201.000, Y -233.200, Z 559.000, A 0.000, B 90.000, C 0.000, E1 0.000, E2 0.0, E3 0.0, E4 0.0, E5 0.0, E6 0.0} C_DIS
LIN {E6POS: X 1201.000, Y -232.200, Z 559.000, A 0.000, B 90.000, C 0.000, E1 0.000, E2 0.0, E3 0.0, E4 0.0, E5 0.0, E6 0.0} C_DIS
LIN {E6POS: X 1201.000, Y -231.200, Z 559.000, A 0.000, B 90.000, C 0.000, E1 0.000, E2 0.0, E3 0.0, E4 0.0, E5 0.0, E6 0.0} C_DIS
LIN {E6POS: X 1201.000, Y -230.200, Z 559.000, A 0.000, B 90.000, C 0.000, E1 0.000, E2 0.0, E3 0.0, E4 0.0, E5 0.0, E6 0.0} C_DIS
LIN {E6POS: X 1201.000, Y -229.200, Z 559.000, A 0.000, B 90.000, C 0.000, E1 0.000, E2 0.0, E3 0.0, E4 0.0, E5 0.0, E6 0.0} C_DIS
LIN {E6POS: X 1201.000, Y -228.200, Z 559.000, A 0.000, B 90.000, C 0.000, E1 0.000, E2 0.0, E3 0.0, E4 0.0, E5 0.0, E6 0.0} C_DIS
LIN {E6POS: X 1201.000, Y -227.200, Z 559.000, A 0.000, B 90.000, C 0.000, E1 0.000, E2 0.0, E3 0.0, E4 0.0, E5 0.0, E6 0.0} C_DIS
LIN {E6POS: X 1201.000, Y -226.200, Z 559.000, A 0.000, B 90.000, C 0.000, E1 0.000, E2 0.0, E3 0.0, E4 0.0, E5 0.0, E6 0.0} C_DIS
LIN {E6POS: X 1201.000, Y -225.200, Z 559.000, A 0.000, B 90.000, C 0.000, E1 0.000, E2 0.0, E3 0.0, E4 0.0, E5 0.0, E6 0.0} C_DIS
LIN {E6POS: X 1201.000, Y -224.200, Z 559.000, A 0.000, B 90.000, C 0.000, E1 0.000, E2 0.0, E3 0.0, E4 0.0, E5 0.0, E6 0.0} C_DIS
LIN {E6POS: X 1201.000, Y -223.200, Z 559.000, A 0.000, B 90.000, C 0.000, E1 0.000, E2 0.0, E3 0.0, E4 0.0, E5 0.0, E6 0.0} C_DIS
LIN {E6POS: X 1201.000, Y -222.200, Z 559.000, A 0.000, B 90.000, C 0.000, E1 0.000, E2 0.0, E3 0.0, E4 0.0, E5 0.0, E6 0.0} C_DIS
LIN {E6POS: X 1201.000, Y -221.200, Z 559.000, A 0.000, B 90.000, C 0.000, E1 0.000, E2 0.0, E3 0.0, E4 0.0, E5 0.0, E6 0.0} C_DIS
LIN {E6POS: X 1201.000, Y -220.200, Z 559.000, A 0.000, B 90.000, C 0.000, E1 0.000, E2 0.0, E3 0.0, E4 0.0, E5 0.0, E6 0.0} C_DIS
LIN {E6POS: X 1201.000, Y -219.200, Z 559.000, A 0.000, B 90.000, C 0.000, E1 0.000, E2 0.0, E3 0.0, E4 0.0, E5 0.0, E6 0.0} C_DIS
LIN {E6POS: X 1201.000, Y -218.200, Z 559.000, A 0.000, B 90.000, C 0.000, E1 0.000, E2 0.0, E3 0.0, E4 0.0, E5 0.0, E6 0.0} C_DIS
LIN {E6POS: X 1201.000, Y -217.200, Z 559.000, A 0.000, B 90.000, C 0.000, E1 0.000, E2 0.0, E3 0.0, E4 0.0, E5 0.0, E6 0.0} C_DIS
LIN {E6POS: X 1201.000, Y -216.200, Z 559.000, A 0.000, B 90.000, C 0.000, E1 0.000, E2 0.0, E3 0.0, E4 0.0, E5 0.0, E6 0.0} C_DIS
LIN {E6POS: X 1201.000, Y -215.200, Z 559.000, A 0.000, B 90.000, C 0.000, E1 0.000, E2 0.0, E3 0.0, E4 0.0, E5 0.0, E6 0.0} C_DIS
LIN {E6POS: X 1201.000, Y -214.200, Z 559.000, A 0.000, B 90.000, C 0.000, E1 0.000, E2 0.0, E3 0.0, E4 0.0, E5 0.0, E6 0.0} C_DIS
LIN {E6POS: X 1201.000, Y -213.200, Z 559.000, A 0.000, B 90.000, C 0.000, E1 0.000, E2 0.0, E3 0.0, E4 0.0, E5 0.0, E6 0.0} C_DIS
LIN {E6POS: X 1201.000, Y -212.200, Z 559.000, A 0.000, B 90.000, C 0.000, E1 0.000, E2 0.0, E3 0.0, E4 0.0, E5 0.0, E6 0.0} C_DIS
LIN {E6POS: X 1201.000, Y -211.200, Z 559.000, A 0.000, B 90.000, C 0.000, E1 0.000, E2 0.0, E3 0.0, E4 0.0, E5 0.0, E6 0.0} C_DIS
LIN {E6POS: X 1201.000, Y -210.200, Z 559.000, A 0.000, B 90.000, C 0.000, E1 0.000, E2 0.0, E3 0.0, E4 0.0, E5 0.0, E6 0.0} C_DIS
LIN {E6POS: X 1201.000, Y -209.200, Z 559.000, A 0.000, B 90.000, C 0.000, E1 0.000, E2 0.0, E3 0.0, E4 0.0, E5 0.0, E6 0.0} C_DIS
LIN {E6POS: X 1201.000, Y -208.200, Z 559.000, A 0.000, B 90.000, C 0.000, E1 0.000, E2 0.0, E3 0.0, E4 0.0, E5 0.0, E6 0.0} C_DIS
LIN {E6POS: X 1201.000, Y -207.200, Z 559.000, A 0.000, B 90.000, C 0.000, E1 0.000, E2 0.0, E3 0.0, E4 0.0, E5 0.0, E6 0.0} C_DIS
LIN {E6POS: X 1201.000, Y -206.200, Z 559.000, A 0.000, B 90.000, C 0.000, E1 0.000, E2 0.0, E3 0.0, E4 0.0, E5 0.0, E6 0.0} C_DIS
LIN {E6POS: X 1201.000, Y -205.200, Z 559.000, A 0.000, B 90.000, C 0.000, E1 0.000, E2 0.0, E3 0.0, E4 0.0, E5 0.0, E6 0.0} C_DIS
LIN {E6POS: X 1201.000, Y -204.200, Z 559.000, A 0.000, B 90.000, C 0.000, E1 0.000, E2 0.0, E3 0.0, E4 0.0, E5 0.0, E6 0.0} C_DIS
LIN {E6POS: X 1201.000, Y -203.200, Z 559.000, A 0.000, B 90.000, C 0.000, E1 0.000, E2 0.0, E3 0.0, E4 0.0, E5 0.0, E6 0.0} C_DIS
LIN {E6POS: X 1201.000, Y -202.200, Z 559.000, A 0.000, B 90.000, C 0.000, E1 0.000, E2 0.0, E3 0.0, E4 0.0, E5 0.0, E6 0.0} C_DIS
LIN {E6POS: X 1201.000, Y -201.200, Z 559.000, A 0.000, B 90.000, C 0.000, E1 0.000, E2 0.0, E3 0.0, E4 0.0, E5 0.0, E6 0.0} C_DIS
LIN {E6POS: X 1201.000, Y -200.200, Z 559.000, A 0.000, B 90.000, C 0.000, E1 0.000, E2 0.0, E3 0.0, E4 0.0, E5 0.0, E6 0.0} C_DIS
LIN {E6POS: X 1201.000, Y -199.200, Z 559.000, A 0.000, B 90.000, C 0.000, E1 0.000, E2 0.0, E3 0.0, E4 0.0, E5 0.0, E6 0.0} C_DIS
LIN {E6POS: X 1201.000, Y -198.200, Z 559.000, A 0.000, B 90.000, C 0.000, E1 0.000, E2 0.0, E3 0.0, E4 0.0, E5 0.0, E6 0.0} C_DIS
LIN {E6POS: X 1201.000, Y -197.200, Z 559.000, A 0.000, B 90.000, C 0.000, E1 0.000, E2 0.0, E3 0.0, E4 0.0, E5 0.0, E6 0.0} C_DIS
LIN {E6POS: X 1201.000, Y -196.200, Z 559.000, A 0.000, B 90.000, C 0.000, E1 0.000, E2 0.0, E3 0.0, E4 0.0, E5 0.0, E6 0.0} C_DIS
LIN {E6POS: X 1201.000, Y -195.200, Z 559.000, A 0.000, B 90.000, C 0.000, E1 0.000, E2 0.0, E3 0.0, E4 0.0, E5 0.0, E6 0.0} C_DIS
LIN {E6POS: X 1201.000, Y -194.200, Z 559.000, A 0.000, B 90.000, C 0.000, E1 0.000, E2 0.0, E3 0.0, E4 0.0, E5 0.0, E6 0.0} C_DIS
LIN {E6POS: X 1201.000, Y -193.200, Z 559.000, A 0.000, B 90.000, C 0.000, E1 0.000, E2 0.0, E3 0.0, E4 0.0, E5 0.0, E6 0.0} C_DIS
LIN {E6POS: X 1201.000, Y -192.200, Z 559.000, A 0.000, B 90.000, C 0.000, E1 0.000, E2 0.0, E3 0.0, E4 0.0, E5 0.0, E6 0.0} C_DIS
LIN {E6POS: X 1201.000, Y -191.200, Z 559.000, A 0.000, B 90.000, C 0.000, E1 0.000, E2 0.0, E3 0.0, E4 0.0, E5 0.0, E6 0.0} C_DIS
LIN {E6POS: X 1201.000, Y -190.200, Z 559.000, A 0.000, B 90.000, C 0.000, E1 0.000, E2 0.0, E3 0.0, E4 0.0, E5 0.0, E6 0.0} C_DIS
LIN {E6POS: X 1201.000, Y -189.200, Z 559.000, A 0.000, B 90.000, C 0.000, E1 0.000, E2 0.0, E3 0.0, E4 0.0, E5 0.0, E6 0.0} C_DIS
LIN {E6POS: X 1201.000, Y -188.200, Z 559.000, A 0.000, B 90.000, C 0.000, E1 0.000, E2 0.0, E3 0.0, E4 0.0, E5 0.0, E6 0.0} C_DIS
LIN {E6POS: X 1201.000, Y -187.200, Z 559.000, A 0.000, B 90.000, C 0.000, E1 0.000, E2 0.0, E3 0.0, E4 0.0, E5 0.0, E6 0.0} C_DIS
LIN {E6POS: X 1201.000, Y -187.200, Z 559.000, A 0.000, B 90.000, C 0.000, E1 0.000, E2 0.0, E3 0.0, E4 0.0, E5 0.0, E6 0.0} C_DIS
LIN {E6POS: X 1200.000, Y -187.200, Z 559.000, A 0.000, B 90.000, C 0.000, E1 0.000, E2 0.0, E3 0.0, E4 0.0, E5 0.0, E6 0.0} C_DIS
LIN {E6POS: X 1199.000, Y -187.200, Z 559.000, A 0.000, B 90.000, C 0.000, E1 0.000, E2 0.0, E3 0.0, E4 0.0, E5 0.0, E6 0.0} C_DIS
LIN {E6POS: X 1198.000, Y -187.200, Z 559.000, A 0.000, B 90.000, C 0.000, E1 0.000, E2 0.0, E3 0.0, E4 0.0, E5 0.0, E6 0.0} C_DIS
LIN {E6POS: X 1197.000, Y -187.200, Z 559.000, A 0.000, B 90.000, C 0.000, E1 0.000, E2 0.0, E3 0.0, E4 0.0, E5 0.0, E6 0.0} C_DIS
LIN {E6POS: X 1196.000, Y -187.200, Z 559.000, A 0.000, B 90.000, C 0.000, E1 0.000, E2 0.0, E3 0.0, E4 0.0, E5 0.0, E6 0.0} C_DIS
LIN {E6POS: X 1196.000, Y -187.200, Z 559.000, A 0.000, B 90.000, C 0.000, E1 0.000, E2 0.0, E3 0.0, E4 0.0, E5 0.0, E6 0.0} C_DIS
LIN {E6POS: X 1196.000, Y -188.200, Z 559.000, A 0.000, B 90.000, C 0.000, E1 0.000, E2 0.0, E3 0.0, E4 0.0, E5 0.0, E6 0.0} C_DIS
LIN {E6POS: X 1196.000, Y -189.200, Z 559.000, A 0.000, B 90.000, C 0.000, E1 0.000, E2 0.0, E3 0.0, E4 0.0, E5 0.0, E6 0.0} C_DIS
LIN {E6POS: X 1196.000, Y -190.200, Z 559.000, A 0.000, B 90.000, C 0.000, E1 0.000, E2 0.0, E3 0.0, E4 0.0, E5 0.0, E6 0.0} C_DIS
LIN {E6POS: X 1196.000, Y -191.200, Z 559.000, A 0.000, B 90.000, C 0.000, E1 0.000, E2 0.0, E3 0.0, E4 0.0, E5 0.0, E6 0.0} C_DIS
LIN {E6POS: X 1196.000, Y -192.200, Z 559.000, A 0.000, B 90.000, C 0.000, E1 0.000, E2 0.0, E3 0.0, E4 0.0, E5 0.0, E6 0.0} C_DIS
LIN {E6POS: X 1196.000, Y -193.200, Z 559.000, A 0.000, B 90.000, C 0.000, E1 0.000, E2 0.0, E3 0.0, E4 0.0, E5 0.0, E6 0.0} C_DIS
LIN {E6POS: X 1196.000, Y -194.200, Z 559.000, A 0.000, B 90.000, C 0.000, E1 0.000, E2 0.0, E3 0.0, E4 0.0, E5 0.0, E6 0.0} C_DIS
LIN {E6POS: X 1196.000, Y -195.200, Z 559.000, A 0.000, B 90.000, C 0.000, E1 0.000, E2 0.0, E3 0.0, E4 0.0, E5 0.0, E6 0.0} C_DIS
LIN {E6POS: X 1196.000, Y -196.200, Z 559.000, A 0.000, B 90.000, C 0.000, E1 0.000, E2 0.0, E3 0.0, E4 0.0, E5 0.0, E6 0.0} C_DIS
LIN {E6POS: X 1196.000, Y -197.200, Z 559.000, A 0.000, B 90.000, C 0.000, E1 0.000, E2 0.0, E3 0.0, E4 0.0, E5 0.0, E6 0.0} C_DIS
LIN {E6POS: X 1196.000, Y -198.200, Z 559.000, A 0.000, B 90.000, C 0.000, E1 0.000, E2 0.0, E3 0.0, E4 0.0, E5 0.0, E6 0.0} C_DIS
LIN {E6POS: X 1196.000, Y -199.200, Z 559.000, A 0.000, B 90.000, C 0.000, E1 0.000, E2 0.0, E3 0.0, E4 0.0, E5 0.0, E6 0.0} C_DIS
LIN {E6POS: X 1196.000, Y -200.200, Z 559.000, A 0.000, B 90.000, C 0.000, E1 0.000, E2 0.0, E3 0.0, E4 0.0, E5 0.0, E6 0.0} C_DIS
LIN {E6POS: X 1196.000, Y -201.200, Z 559.000, A 0.000, B 90.000, C 0.000, E1 0.000, E2 0.0, E3 0.0, E4 0.0, E5 0.0, E6 0.0} C_DIS
LIN {E6POS: X 1196.000, Y -202.200, Z 559.000, A 0.000, B 90.000, C 0.000, E1 0.000, E2 0.0, E3 0.0, E4 0.0, E5 0.0, E6 0.0} C_DIS
LIN {E6POS: X 1196.000, Y -203.200, Z 559.000, A 0.000, B 90.000, C 0.000, E1 0.000, E2 0.0, E3 0.0, E4 0.0, E5 0.0, E6 0.0} C_DIS
LIN {E6POS: X 1196.000, Y -204.200, Z 559.000, A 0.000, B 90.000, C 0.000, E1 0.000, E2 0.0, E3 0.0, E4 0.0, E5 0.0, E6 0.0} C_DIS
LIN {E6POS: X 1196.000, Y -205.200, Z 559.000, A 0.000, B 90.000, C 0.000, E1 0.000, E2 0.0, E3 0.0, E4 0.0, E5 0.0, E6 0.0} C_DIS
LIN {E6POS: X 1196.000, Y -206.200, Z 559.000, A 0.000, B 90.000, C 0.000, E1 0.000, E2 0.0, E3 0.0, E4 0.0, E5 0.0, E6 0.0} C_DIS
LIN {E6POS: X 1196.000, Y -207.200, Z 559.000, A 0.000, B 90.000, C 0.000, E1 0.000, E2 0.0, E3 0.0, E4 0.0, E5 0.0, E6 0.0} C_DIS
LIN {E6POS: X 1196.000, Y -208.200, Z 559.000, A 0.000, B 90.000, C 0.000, E1 0.000, E2 0.0, E3 0.0, E4 0.0, E5 0.0, E6 0.0} C_DIS
LIN {E6POS: X 1196.000, Y -209.200, Z 559.000, A 0.000, B 90.000, C 0.000, E1 0.000, E2 0.0, E3 0.0, E4 0.0, E5 0.0, E6 0.0} C_DIS
LIN {E6POS: X 1196.000, Y -210.200, Z 559.000, A 0.000, B 90.000, C 0.000, E1 0.000, E2 0.0, E3 0.0, E4 0.0, E5 0.0, E6 0.0} C_DIS
LIN {E6POS: X 1196.000, Y -211.200, Z 559.000, A 0.000, B 90.000, C 0.000, E1 0.000, E2 0.0, E3 0.0, E4 0.0, E5 0.0, E6 0.0} C_DIS
LIN {E6POS: X 1196.000, Y -212.200, Z 559.000, A 0.000, B 90.000, C 0.000, E1 0.000, E2 0.0, E3 0.0, E4 0.0, E5 0.0, E6 0.0} C_DIS
LIN {E6POS: X 1196.000, Y -213.200, Z 559.000, A 0.000, B 90.000, C 0.000, E1 0.000, E2 0.0, E3 0.0, E4 0.0, E5 0.0, E6 0.0} C_DIS
LIN {E6POS: X 1196.000, Y -214.200, Z 559.000, A 0.000, B 90.000, C 0.000, E1 0.000, E2 0.0, E3 0.0, E4 0.0, E5 0.0, E6 0.0} C_DIS
LIN {E6POS: X 1196.000, Y -215.200, Z 559.000, A 0.000, B 90.000, C 0.000, E1 0.000, E2 0.0, E3 0.0, E4 0.0, E5 0.0, E6 0.0} C_DIS
LIN {E6POS: X 1196.000, Y -216.200, Z 559.000, A 0.000, B 90.000, C 0.000, E1 0.000, E2 0.0, E3 0.0, E4 0.0, E5 0.0, E6 0.0} C_DIS
LIN {E6POS: X 1196.000, Y -217.200, Z 559.000, A 0.000, B 90.000, C 0.000, E1 0.000, E2 0.0, E3 0.0, E4 0.0, E5 0.0, E6 0.0} C_DIS
LIN {E6POS: X 1196.000, Y -218.200, Z 559.000, A 0.000, B 90.000, C 0.000, E1 0.000, E2 0.0, E3 0.0, E4 0.0, E5 0.0, E6 0.0} C_DIS
LIN {E6POS: X 1196.000, Y -219.200, Z 559.000, A 0.000, B 90.000, C 0.000, E1 0.000, E2 0.0, E3 0.0, E4 0.0, E5 0.0, E6 0.0} C_DIS
LIN {E6POS: X 1196.000, Y -220.200, Z 559.000, A 0.000, B 90.000, C 0.000, E1 0.000, E2 0.0, E3 0.0, E4 0.0, E5 0.0, E6 0.0} C_DIS
LIN {E6POS: X 1196.000, Y -221.200, Z 559.000, A 0.000, B 90.000, C 0.000, E1 0.000, E2 0.0, E3 0.0, E4 0.0, E5 0.0, E6 0.0} C_DIS
LIN {E6POS: X 1196.000, Y -222.200, Z 559.000, A 0.000, B 90.000, C 0.000, E1 0.000, E2 0.0, E3 0.0, E4 0.0, E5 0.0, E6 0.0} C_DIS
LIN {E6POS: X 1196.000, Y -223.200, Z 559.000, A 0.000, B 90.000, C 0.000, E1 0.000, E2 0.0, E3 0.0, E4 0.0, E5 0.0, E6 0.0} C_DIS
LIN {E6POS: X 1196.000, Y -224.200, Z 559.000, A 0.000, B 90.000, C 0.000, E1 0.000, E2 0.0, E3 0.0, E4 0.0, E5 0.0, E6 0.0} C_DIS
LIN {E6POS: X 1196.000, Y -225.200, Z 559.000, A 0.000, B 90.000, C 0.000, E1 0.000, E2 0.0, E3 0.0, E4 0.0, E5 0.0, E6 0.0} C_DIS
LIN {E6POS: X 1196.000, Y -226.200, Z 559.000, A 0.000, B 90.000, C 0.000, E1 0.000, E2 0.0, E3 0.0, E4 0.0, E5 0.0, E6 0.0} C_DIS
LIN {E6POS: X 1196.000, Y -227.200, Z 559.000, A 0.000, B 90.000, C 0.000, E1 0.000, E2 0.0, E3 0.0, E4 0.0, E5 0.0, E6 0.0} C_DIS
LIN {E6POS: X 1196.000, Y -228.200, Z 559.000, A 0.000, B 90.000, C 0.000, E1 0.000, E2 0.0, E3 0.0, E4 0.0, E5 0.0, E6 0.0} C_DIS
LIN {E6POS: X 1196.000, Y -229.200, Z 559.000, A 0.000, B 90.000, C 0.000, E1 0.000, E2 0.0, E3 0.0, E4 0.0, E5 0.0, E6 0.0} C_DIS
LIN {E6POS: X 1196.000, Y -230.200, Z 559.000, A 0.000, B 90.000, C 0.000, E1 0.000, E2 0.0, E3 0.0, E4 0.0, E5 0.0, E6 0.0} C_DIS
LIN {E6POS: X 1196.000, Y -231.200, Z 559.000, A 0.000, B 90.000, C 0.000, E1 0.000, E2 0.0, E3 0.0, E4 0.0, E5 0.0, E6 0.0} C_DIS
LIN {E6POS: X 1196.000, Y -232.200, Z 559.000, A 0.000, B 90.000, C 0.000, E1 0.000, E2 0.0, E3 0.0, E4 0.0, E5 0.0, E6 0.0} C_DIS
LIN {E6POS: X 1196.000, Y -233.200, Z 559.000, A 0.000, B 90.000, C 0.000, E1 0.000, E2 0.0, E3 0.0, E4 0.0, E5 0.0, E6 0.0} C_DIS
LIN {E6POS: X 1196.000, Y -234.200, Z 559.000, A 0.000, B 90.000, C 0.000, E1 0.000, E2 0.0, E3 0.0, E4 0.0, E5 0.0, E6 0.0} C_DIS
LIN {E6POS: X 1196.000, Y -235.200, Z 559.000, A 0.000, B 90.000, C 0.000, E1 0.000, E2 0.0, E3 0.0, E4 0.0, E5 0.0, E6 0.0} C_DIS
LIN {E6POS: X 1196.000, Y -236.200, Z 559.000, A 0.000, B 90.000, C 0.000, E1 0.000, E2 0.0, E3 0.0, E4 0.0, E5 0.0, E6 0.0} C_DIS
LIN {E6POS: X 1196.000, Y -237.200, Z 559.000, A 0.000, B 90.000, C 0.000, E1 0.000, E2 0.0, E3 0.0, E4 0.0, E5 0.0, E6 0.0} C_DIS
LIN {E6POS: X 1196.000, Y -237.200, Z 560.000, A 0.000, B 90.000, C 0.000, E1 0.000, E2 0.0, E3 0.0, E4 0.0, E5 0.0, E6 0.0} C_DIS
LIN {E6POS: X 1197.000, Y -237.200, Z 560.000, A 0.000, B 90.000, C 0.000, E1 0.000, E2 0.0, E3 0.0, E4 0.0, E5 0.0, E6 0.0} C_DIS
LIN {E6POS: X 1198.000, Y -237.200, Z 560.000, A 0.000, B 90.000, C 0.000, E1 0.000, E2 0.0, E3 0.0, E4 0.0, E5 0.0, E6 0.0} C_DIS
LIN {E6POS: X 1199.000, Y -237.200, Z 560.000, A 0.000, B 90.000, C 0.000, E1 0.000, E2 0.0, E3 0.0, E4 0.0, E5 0.0, E6 0.0} C_DIS
LIN {E6POS: X 1200.000, Y -237.200, Z 560.000, A 0.000, B 90.000, C 0.000, E1 0.000, E2 0.0, E3 0.0, E4 0.0, E5 0.0, E6 0.0} C_DIS
LIN {E6POS: X 1201.000, Y -237.200, Z 560.000, A 0.000, B 90.000, C 0.000, E1 0.000, E2 0.0, E3 0.0, E4 0.0, E5 0.0, E6 0.0} C_DIS
LIN {E6POS: X 1201.000, Y -237.200, Z 560.000, A 0.000, B 90.000, C 0.000, E1 0.000, E2 0.0, E3 0.0, E4 0.0, E5 0.0, E6 0.0} C_DIS
LIN {E6POS: X 1201.000, Y -236.200, Z 560.000, A 0.000, B 90.000, C 0.000, E1 0.000, E2 0.0, E3 0.0, E4 0.0, E5 0.0, E6 0.0} C_DIS
LIN {E6POS: X 1201.000, Y -235.200, Z 560.000, A 0.000, B 90.000, C 0.000, E1 0.000, E2 0.0, E3 0.0, E4 0.0, E5 0.0, E6 0.0} C_DIS
LIN {E6POS: X 1201.000, Y -234.200, Z 560.000, A 0.000, B 90.000, C 0.000, E1 0.000, E2 0.0, E3 0.0, E4 0.0, E5 0.0, E6 0.0} C_DIS
LIN {E6POS: X 1201.000, Y -233.200, Z 560.000, A 0.000, B 90.000, C 0.000, E1 0.000, E2 0.0, E3 0.0, E4 0.0, E5 0.0, E6 0.0} C_DIS
LIN {E6POS: X 1201.000, Y -232.200, Z 560.000, A 0.000, B 90.000, C 0.000, E1 0.000, E2 0.0, E3 0.0, E4 0.0, E5 0.0, E6 0.0} C_DIS
LIN {E6POS: X 1201.000, Y -231.200, Z 560.000, A 0.000, B 90.000, C 0.000, E1 0.000, E2 0.0, E3 0.0, E4 0.0, E5 0.0, E6 0.0} C_DIS
LIN {E6POS: X 1201.000, Y -230.200, Z 560.000, A 0.000, B 90.000, C 0.000, E1 0.000, E2 0.0, E3 0.0, E4 0.0, E5 0.0, E6 0.0} C_DIS
LIN {E6POS: X 1201.000, Y -229.200, Z 560.000, A 0.000, B 90.000, C 0.000, E1 0.000, E2 0.0, E3 0.0, E4 0.0, E5 0.0, E6 0.0} C_DIS
LIN {E6POS: X 1201.000, Y -228.200, Z 560.000, A 0.000, B 90.000, C 0.000, E1 0.000, E2 0.0, E3 0.0, E4 0.0, E5 0.0, E6 0.0} C_DIS
